LIN {X 0,Y 425.396,Z 103.811,A -85,B 0,C 180,E1 -9909.51,E2 -9909.51} C_VEL
LIN {X 0,Y 425.389,Z 103.807,A -85,B 0,C 180,E1 -9912.904,E2 -9912.904} C_VEL
LIN {X 0,Y 425.357,Z 103.809,A -85,B 0,C 180,E1 -9916.605,E2 -9916.605} C_VEL
LIN {X 0,Y 425.324,Z 103.816,A -85,B 0,C 180,E1 -9919.636,E2 -9919.636} C_VEL
LIN {X 0,Y 425.303,Z 103.821,A -85,B 0,C 180,E1 -9923.365,E2 -9923.365} C_VEL
LIN {X 0,Y 425.343,Z 103.814,A -85,B 0,C 180,E1 -9926.844,E2 -9926.844} C_VEL
LIN {X 0,Y 425.287,Z 103.819,A -85,B 0,C 180,E1 -9929.72,E2 -9929.72} C_VEL
LIN {X 0,Y 425.278,Z 103.826,A -85,B 0,C 180,E1 -9933.048,E2 -9933.048} C_VEL
LIN {X 0,Y 425.281,Z 103.818,A -85,B 0,C 180,E1 -9935.93,E2 -9935.93} C_VEL
LIN {X 0,Y 425.297,Z 103.823,A -85,B 0,C 180,E1 -9939.044,E2 -9939.044} C_VEL
LIN {X 0,Y 425.275,Z 103.824,A -85,B 0,C 180,E1 -9942.653,E2 -9942.653} C_VEL
LIN {X 0,Y 425.265,Z 103.821,A -85,B 0,C 180,E1 -9946.046,E2 -9946.046} C_VEL
LIN {X 0,Y 425.301,Z 103.821,A -85,B 0,C 180,E1 -9948.626,E2 -9948.626} C_VEL
LIN {X 0,Y 425.313,Z 103.818,A -85,B 0,C 180,E1 -9951.104,E2 -9951.104} C_VEL
LIN {X 0,Y 425.296,Z 103.824,A -85,B 0,C 180,E1 -9954.665,E2 -9954.665} C_VEL
LIN {X 0,Y 425.263,Z 103.822,A -85,B 0,C 180,E1 -9958.074,E2 -9958.074} C_VEL
LIN {X 0,Y 425.329,Z 103.813,A -85,B 0,C 180,E1 -9961.369,E2 -9961.369} C_VEL
LIN {X 0,Y 425.295,Z 103.824,A -85,B 0,C 180,E1 -9964.555,E2 -9964.555} C_VEL
LIN {X 0,Y 425.286,Z 103.818,A -85,B 0,C 180,E1 -9967.662,E2 -9967.662} C_VEL
LIN {X 0,Y 425.364,Z 103.812,A -85,B 0,C 180,E1 -9970.705,E2 -9970.705} C_VEL
LIN {X 0,Y 425.388,Z 103.806,A -85,B 0,C 180,E1 -9973.689,E2 -9973.689} C_VEL
LIN {X 0,Y 425.412,Z 103.803,A -85,B 0,C 180,E1 -9977.599,E2 -9977.599} C_VEL
LIN {X 0,Y 425.443,Z 103.799,A -85,B 0,C 180,E1 -9981.451,E2 -9981.451} C_VEL
LIN {X 0,Y 425.554,Z 103.79,A -85,B 0,C 180,E1 -9984.314,E2 -9984.314} C_VEL
LIN {X 0,Y 425.574,Z 103.79,A -85,B 0,C 180,E1 -9988.108,E2 -9988.108} C_VEL
LIN {X 0,Y 425.702,Z 103.773,A -85,B 0,C 180,E1 -9990.001,E2 -9990.001} C_VEL
LIN {X 0,Y 425.546,Z 103.786,A -85,B 0,C 180,E1 -9992.841,E2 -9992.841} C_VEL
LIN {X 0,Y 425.532,Z 103.788,A -85,B 0,C 180,E1 -9996.639,E2 -9996.639} C_VEL
LIN {X 0,Y 425.404,Z 103.804,A -85,B 0,C 180,E1 -9999.153,E2 -9999.153} C_VEL
LIN {X 0,Y 424.732,Z 103.894,A -85,B 0,C 180,E1 -9999.943,E2 -9999.943} C_VEL
LIN {X 0,Y 421.884,Z 104.243,A -85,B 0,C 180,E1 -10001.226,E2 -10001.226} C_VEL
LIN {X 0,Y 419.468,Z 104.545,A -85,B 0,C 180,E1 -10002.262,E2 -10002.262} C_VEL
LIN {X 0,Y 418.417,Z 104.674,A -85,B 0,C 180,E1 -10003.063,E2 -10003.063} C_VEL
LIN {X 0,Y 418.324,Z 104.687,A -85,B 0,C 180,E1 -10003.334,E2 -10003.334} C_VEL
LIN {X 0,Y 418.315,Z 104.686,A -85,B 0,C 180,E1 -10006.736,E2 -10006.736} C_VEL
LIN {X 0,Y 418.273,Z 104.698,A -85,B 0,C 180,E1 -10009.791,E2 -10009.791} C_VEL
LIN {X 0,Y 418.24,Z 104.696,A -85,B 0,C 180,E1 -10012.737,E2 -10012.737} C_VEL
LIN {X 0,Y 418.271,Z 104.695,A -85,B 0,C 180,E1 -10015.905,E2 -10015.905} C_VEL
LIN {X 0,Y 418.267,Z 104.695,A -85,B 0,C 180,E1 -10019.162,E2 -10019.162} C_VEL
LIN {X 0,Y 418.26,Z 104.694,A -85,B 0,C 180,E1 -10022.844,E2 -10022.844} C_VEL
LIN {X 0,Y 418.247,Z 104.695,A -85,B 0,C 180,E1 -10026.238,E2 -10026.238} C_VEL
LIN {X 0,Y 418.254,Z 104.697,A -85,B 0,C 180,E1 -10029.682,E2 -10029.682} C_VEL
LIN {X 0,Y 418.234,Z 104.696,A -85,B 0,C 180,E1 -10032.322,E2 -10032.322} C_VEL
LIN {X 0,Y 418.241,Z 104.701,A -85,B 0,C 180,E1 -10035.109,E2 -10035.109} C_VEL
LIN {X 0,Y 418.243,Z 104.697,A -85,B 0,C 180,E1 -10037.767,E2 -10037.767} C_VEL
LIN {X 0,Y 418.252,Z 104.696,A -85,B 0,C 180,E1 -10040.62,E2 -10040.62} C_VEL
LIN {X 0,Y 418.247,Z 104.699,A -85,B 0,C 180,E1 -10043.976,E2 -10043.976} C_VEL
LIN {X 0,Y 418.261,Z 104.698,A -85,B 0,C 180,E1 -10047.156,E2 -10047.156} C_VEL
LIN {X 0,Y 418.256,Z 104.744,A -85,B 0,C 180,E1 -10047.691,E2 -10047.691} C_VEL
LIN {X 0,Y 419.311,Z 107.662,A -85,B 0,C 180,E1 -10047.841,E2 -10047.841} C_VEL
LIN {X 0,Y 434.601,Z 137.945,A -85,B 0,C 180,E1 -10049.622,E2 -10049.622} C_VEL
LIN {X 0,Y 430.278,Z 282.426,A -85,B 0,C 180,E1 -10052.554,E2 -10052.554} C_VEL
LIN {X 0,Y 429.662,Z 301.528,A -85,B 0,C 180,E1 -10053.005,E2 -10053.005} C_VEL
LIN {X 0,Y 428.924,Z 318.826,A -85,B 0,C 180,E1 -10053.612,E2 -10053.612} C_VEL
LIN {X 0,Y 427.987,Z 335.334,A -85,B 0,C 180,E1 -10054.386,E2 -10054.386} C_VEL
LIN {X 0,Y 427.104,Z 349.564,A -85,B 0,C 180,E1 -10055.22,E2 -10055.22} C_VEL
LIN {X 0,Y 425.867,Z 364.452,A -85,B 0,C 180,E1 -10056.281,E2 -10056.281} C_VEL
LIN {X 0,Y 424.626,Z 378.646,A -85,B 0,C 180,E1 -10057.496,E2 -10057.496} C_VEL
LIN {X 0,Y 423.459,Z 391.882,A -85,B 0,C 180,E1 -10058.84,E2 -10058.84} C_VEL
LIN {X 0,Y 422.25,Z 404.22,A -85,B 0,C 180,E1 -10060.303,E2 -10060.303} C_VEL
LIN {X 0,Y 421.134,Z 416.557,A -85,B 0,C 180,E1 -10062.034,E2 -10062.034} C_VEL
LIN {X 0,Y 420.175,Z 426.779,A -85,B 0,C 180,E1 -10063.73,E2 -10063.73} C_VEL
LIN {X 0,Y 419.373,Z 435.593,A -85,B 0,C 180,E1 -10065.441,E2 -10065.441} C_VEL
LIN {X 0,Y 418.682,Z 444.113,A -85,B 0,C 180,E1 -10067.396,E2 -10067.396} C_VEL
LIN {X 0,Y 418.129,Z 451.181,A -85,B 0,C 180,E1 -10069.345,E2 -10069.345} C_VEL
LIN {X 0,Y 417.81,Z 456.853,A -85,B 0,C 180,E1 -10071.292,E2 -10071.292} C_VEL
LIN {X 0,Y 417.603,Z 461.379,A -85,B 0,C 180,E1 -10073.234,E2 -10073.234} C_VEL
LIN {X 0,Y 417.363,Z 464.808,A -85,B 0,C 180,E1 -10075.17,E2 -10075.17} C_VEL
LIN {X 0,Y 417.372,Z 467.119,A -85,B 0,C 180,E1 -10077.104,E2 -10077.104} C_VEL
LIN {X 0,Y 417.219,Z 468.502,A -85,B 0,C 180,E1 -10079.035,E2 -10079.035} C_VEL
LIN {X 0,Y 417.221,Z 468.775,A -85,B 0,C 180,E1 -10080.965,E2 -10080.965} C_VEL
LIN {X 0,Y 417.491,Z 468.097,A -85,B 0,C 180,E1 -10082.895,E2 -10082.895} C_VEL
LIN {X 0,Y 417.563,Z 466.374,A -85,B 0,C 180,E1 -10084.827,E2 -10084.827} C_VEL
LIN {X 0,Y 417.796,Z 463.165,A -85,B 0,C 180,E1 -10087.03,E2 -10087.03} C_VEL
LIN {X 0,Y 418.18,Z 458.676,A -85,B 0,C 180,E1 -10089.187,E2 -10089.187} C_VEL
LIN {X 0,Y 418.736,Z 453.445,A -85,B 0,C 180,E1 -10091.129,E2 -10091.129} C_VEL
LIN {X 0,Y 419.34,Z 446.871,A -85,B 0,C 180,E1 -10093.077,E2 -10093.077} C_VEL
LIN {X 0,Y 420.259,Z 438.912,A -85,B 0,C 180,E1 -10095.023,E2 -10095.023} C_VEL
LIN {X 0,Y 421.348,Z 429.335,A -85,B 0,C 180,E1 -10096.971,E2 -10096.971} C_VEL
LIN {X 0,Y 422.531,Z 419.574,A -85,B 0,C 180,E1 -10098.649,E2 -10098.649} C_VEL
LIN {X 0,Y 423.927,Z 407.703,A -85,B 0,C 180,E1 -10100.374,E2 -10100.374} C_VEL
LIN {X 0,Y 425.482,Z 393.99,A -85,B 0,C 180,E1 -10102.044,E2 -10102.044} C_VEL
LIN {X 0,Y 427.128,Z 379.392,A -85,B 0,C 180,E1 -10103.516,E2 -10103.516} C_VEL
LIN {X 0,Y 428.551,Z 365.071,A -85,B 0,C 180,E1 -10104.72,E2 -10104.72} C_VEL
LIN {X 0,Y 429.738,Z 351.619,A -85,B 0,C 180,E1 -10105.671,E2 -10105.671} C_VEL
LIN {X 0,Y 431.066,Z 334.858,A -85,B 0,C 180,E1 -10106.638,E2 -10106.638} C_VEL
LIN {X 0,Y 432.092,Z 318.332,A -85,B 0,C 180,E1 -10107.387,E2 -10107.387} C_VEL
LIN {X 0,Y 432.944,Z 301.612,A -85,B 0,C 180,E1 -10107.952,E2 -10107.952} C_VEL
LIN {X 0,Y 437.02,Z 225.54,A -85,B 0,C 180,E1 -10109.847,E2 -10109.847} C_VEL
LIN {X 0,Y 442.861,Z 147.406,A -85,B 0,C 180,E1 -10111.912,E2 -10111.912} C_VEL
LIN {X 0,Y 443.142,Z 143.294,A -85,B 0,C 180,E1 -10112.033,E2 -10112.033} C_VEL
LIN {X 0,Y 438.622,Z 134.82,A -85,B 0,C 180,E1 -10113.056,E2 -10113.056} C_VEL
LIN {X 0,Y 434.512,Z 127.988,A -85,B 0,C 180,E1 -10114.077,E2 -10114.077} C_VEL
LIN {X 0,Y 431.135,Z 123.216,A -85,B 0,C 180,E1 -10114.973,E2 -10114.973} C_VEL
LIN {X 0,Y 427.821,Z 118.988,A -85,B 0,C 180,E1 -10115.948,E2 -10115.948} C_VEL
LIN {X 0,Y 422.509,Z 113.054,A -85,B 0,C 180,E1 -10117.822,E2 -10117.822} C_VEL
LIN {X 0,Y 421.55,Z 111.994,A -85,B 0,C 180,E1 -10118.3,E2 -10118.3} C_VEL
LIN {X 0,Y 420.598,Z 109.865,A -85,B 0,C 180,E1 -10120.668,E2 -10120.668} C_VEL
LIN {X 0,Y 420.52,Z 109.347,A -85,B 0,C 180,E1 -10121.952,E2 -10121.952} C_VEL
LIN {X 0,Y 420.653,Z 110.069,A -85,B 0,C 180,E1 -10124.075,E2 -10124.075} C_VEL
LIN {X 0,Y 421.369,Z 111.749,A -85,B 0,C 180,E1 -10125.823,E2 -10125.823} C_VEL
LIN {X 0,Y 422.878,Z 114.606,A -85,B 0,C 180,E1 -10127.738,E2 -10127.738} C_VEL
LIN {X 0,Y 424.752,Z 118.675,A -85,B 0,C 180,E1 -10129.563,E2 -10129.563} C_VEL
LIN {X 0,Y 426.873,Z 123.698,A -85,B 0,C 180,E1 -10131.271,E2 -10131.271} C_VEL
LIN {X 0,Y 429.708,Z 131.075,A -85,B 0,C 180,E1 -10133.264,E2 -10133.264} C_VEL
LIN {X 0,Y 431.088,Z 134.99,A -85,B 0,C 180,E1 -10134.126,E2 -10134.126} C_VEL
LIN {X 0,Y 435.256,Z 143.345,A -85,B 0,C 180,E1 -10135.282,E2 -10135.282} C_VEL
LIN {X 0,Y 437.837,Z 149.267,A -85,B 0,C 180,E1 -10135.963,E2 -10135.963} C_VEL
LIN {X 0,Y 439.521,Z 164.422,A -85,B 0,C 180,E1 -10136.829,E2 -10136.829} C_VEL
LIN {X 0,Y 440.924,Z 183.827,A -85,B 0,C 180,E1 -10137.748,E2 -10137.748} C_VEL
LIN {X 0,Y 441.044,Z 188.8,A -85,B 0,C 180,E1 -10137.944,E2 -10137.944} C_VEL
LIN {X 0,Y 436.113,Z 262.024,A -85,B 0,C 180,E1 -10139.828,E2 -10139.828} C_VEL
LIN {X 0,Y 432.849,Z 326.235,A -85,B 0,C 180,E1 -10141.39,E2 -10141.39} C_VEL
LIN {X 0,Y 431.402,Z 356.177,A -85,B 0,C 180,E1 -10142.137,E2 -10142.137} C_VEL
LIN {X 0,Y 429.892,Z 374.913,A -85,B 0,C 180,E1 -10142.79,E2 -10142.79} C_VEL
LIN {X 0,Y 428.455,Z 391.774,A -85,B 0,C 180,E1 -10143.58,E2 -10143.58} C_VEL
LIN {X 0,Y 426.854,Z 407.978,A -85,B 0,C 180,E1 -10144.523,E2 -10144.523} C_VEL
LIN {X 0,Y 425.144,Z 424.654,A -85,B 0,C 180,E1 -10145.719,E2 -10145.719} C_VEL
LIN {X 0,Y 423.574,Z 440.021,A -85,B 0,C 180,E1 -10147.05,E2 -10147.05} C_VEL
LIN {X 0,Y 422.113,Z 454.241,A -85,B 0,C 180,E1 -10148.512,E2 -10148.512} C_VEL
LIN {X 0,Y 420.719,Z 468.305,A -85,B 0,C 180,E1 -10150.228,E2 -10150.228} C_VEL
LIN {X 0,Y 419.628,Z 480.238,A -85,B 0,C 180,E1 -10151.95,E2 -10151.95} C_VEL
LIN {X 0,Y 418.772,Z 490.482,A -85,B 0,C 180,E1 -10153.673,E2 -10153.673} C_VEL
LIN {X 0,Y 418.162,Z 499.345,A -85,B 0,C 180,E1 -10155.397,E2 -10155.397} C_VEL
LIN {X 0,Y 417.694,Z 507.935,A -85,B 0,C 180,E1 -10157.392,E2 -10157.392} C_VEL
LIN {X 0,Y 417.361,Z 514.845,A -85,B 0,C 180,E1 -10159.325,E2 -10159.325} C_VEL
LIN {X 0,Y 417.231,Z 520.598,A -85,B 0,C 180,E1 -10161.28,E2 -10161.28} C_VEL
LIN {X 0,Y 417.307,Z 525.707,A -85,B 0,C 180,E1 -10163.531,E2 -10163.531} C_VEL
LIN {X 0,Y 417.187,Z 529.663,A -85,B 0,C 180,E1 -10166.136,E2 -10166.136} C_VEL
LIN {X 0,Y 417.281,Z 531.295,A -85,B 0,C 180,E1 -10168.069,E2 -10168.069} C_VEL
LIN {X 0,Y 417.174,Z 531.882,A -85,B 0,C 180,E1 -10169.999,E2 -10169.999} C_VEL
LIN {X 0,Y 417.294,Z 531.377,A -85,B 0,C 180,E1 -10171.93,E2 -10171.93} C_VEL
LIN {X 0,Y 417.191,Z 529.776,A -85,B 0,C 180,E1 -10173.863,E2 -10173.863} C_VEL
LIN {X 0,Y 417.217,Z 527.105,A -85,B 0,C 180,E1 -10175.8,E2 -10175.8} C_VEL
LIN {X 0,Y 417.222,Z 523.234,A -85,B 0,C 180,E1 -10177.744,E2 -10177.744} C_VEL
LIN {X 0,Y 417.231,Z 518.213,A -85,B 0,C 180,E1 -10179.697,E2 -10179.697} C_VEL
LIN {X 0,Y 417.51,Z 511.87,A -85,B 0,C 180,E1 -10181.653,E2 -10181.653} C_VEL
LIN {X 0,Y 417.894,Z 504.094,A -85,B 0,C 180,E1 -10183.617,E2 -10183.617} C_VEL
LIN {X 0,Y 418.57,Z 494.75,A -85,B 0,C 180,E1 -10185.583,E2 -10185.583} C_VEL
LIN {X 0,Y 419.329,Z 484.83,A -85,B 0,C 180,E1 -10187.349,E2 -10187.349} C_VEL
LIN {X 0,Y 420.25,Z 473.712,A -85,B 0,C 180,E1 -10189.032,E2 -10189.032} C_VEL
LIN {X 0,Y 421.454,Z 461.108,A -85,B 0,C 180,E1 -10190.648,E2 -10190.648} C_VEL
LIN {X 0,Y 422.725,Z 447.832,A -85,B 0,C 180,E1 -10192.095,E2 -10192.095} C_VEL
LIN {X 0,Y 424.021,Z 433.225,A -85,B 0,C 180,E1 -10193.439,E2 -10193.439} C_VEL
LIN {X 0,Y 425.488,Z 417.781,A -85,B 0,C 180,E1 -10194.615,E2 -10194.615} C_VEL
LIN {X 0,Y 426.713,Z 402.934,A -85,B 0,C 180,E1 -10195.55,E2 -10195.55} C_VEL
LIN {X 0,Y 427.953,Z 386.241,A -85,B 0,C 180,E1 -10196.386,E2 -10196.386} C_VEL
LIN {X 0,Y 429.007,Z 368.899,A -85,B 0,C 180,E1 -10197.038,E2 -10197.038} C_VEL
LIN {X 0,Y 429.847,Z 351.558,A -85,B 0,C 180,E1 -10197.487,E2 -10197.487} C_VEL
LIN {X 0,Y 434.839,Z 186.692,A -85,B 0,C 180,E1 -10200.839,E2 -10200.839} C_VEL
LIN {X 0,Y 429.925,Z 149.859,A -85,B 0,C 180,E1 -10202.053,E2 -10202.053} C_VEL
LIN {X 0,Y 430.466,Z 143.061,A -85,B 0,C 180,E1 -10202.756,E2 -10202.756} C_VEL
LIN {X 0,Y 426.121,Z 128.649,A -85,B 0,C 180,E1 -10204.656,E2 -10204.656} C_VEL
LIN {X 0,Y 419.021,Z 107.167,A -85,B 0,C 180,E1 -10207.659,E2 -10207.659} C_VEL
LIN {X 0,Y 418.224,Z 104.704,A -85,B 0,C 180,E1 -10208.033,E2 -10208.033} C_VEL
LIN {X 0,Y 418.257,Z 104.699,A -85,B 0,C 180,E1 -10210.943,E2 -10210.943} C_VEL
LIN {X 0,Y 418.264,Z 104.696,A -85,B 0,C 180,E1 -10213.737,E2 -10213.737} C_VEL
LIN {X 0,Y 418.207,Z 104.706,A -85,B 0,C 180,E1 -10216.449,E2 -10216.449} C_VEL
LIN {X 0,Y 418.22,Z 104.698,A -85,B 0,C 180,E1 -10219.13,E2 -10219.13} C_VEL
LIN {X 0,Y 418.23,Z 104.703,A -85,B 0,C 180,E1 -10222.165,E2 -10222.165} C_VEL
LIN {X 0,Y 418.261,Z 104.693,A -85,B 0,C 180,E1 -10225.419,E2 -10225.419} C_VEL
LIN {X 0,Y 418.215,Z 104.701,A -85,B 0,C 180,E1 -10228.604,E2 -10228.604} C_VEL
LIN {X 0,Y 418.29,Z 104.694,A -85,B 0,C 180,E1 -10231.937,E2 -10231.937} C_VEL
LIN {X 0,Y 418.285,Z 104.69,A -85,B 0,C 180,E1 -10235.163,E2 -10235.163} C_VEL
LIN {X 0,Y 418.23,Z 104.701,A -85,B 0,C 180,E1 -10238.304,E2 -10238.304} C_VEL
LIN {X 0,Y 418.279,Z 104.692,A -85,B 0,C 180,E1 -10241.383,E2 -10241.383} C_VEL
LIN {X 0,Y 418.306,Z 104.689,A -85,B 0,C 180,E1 -10244.406,E2 -10244.406} C_VEL
LIN {X 0,Y 418.365,Z 104.682,A -85,B 0,C 180,E1 -10247.386,E2 -10247.386} C_VEL
LIN {X 0,Y 418.355,Z 104.683,A -85,B 0,C 180,E1 -10250.329,E2 -10250.329} C_VEL
LIN {X 0,Y 418.489,Z 104.666,A -85,B 0,C 180,E1 -10253.249,E2 -10253.249} C_VEL
LIN {X 0,Y 418.336,Z 104.685,A -85,B 0,C 180,E1 -10255.182,E2 -10255.182} C_VEL
LIN {X 0,Y 418.54,Z 104.661,A -85,B 0,C 180,E1 -10258.076,E2 -10258.076} C_VEL
LIN {X 0,Y 418.668,Z 104.645,A -85,B 0,C 180,E1 -10260,E2 -10260} C_VEL
LIN {X 0,Y 418.506,Z 104.663,A -85,B 0,C 180,E1 -10262.888,E2 -10262.888} C_VEL
LIN {X 0,Y 418.489,Z 104.665,A -85,B 0,C 180,E1 -10266.751,E2 -10266.751} C_VEL
LIN {X 0,Y 418.396,Z 104.677,A -85,B 0,C 180,E1 -10268.695,E2 -10268.695} C_VEL
LIN {X 0,Y 418.312,Z 104.691,A -85,B 0,C 180,E1 -10271.631,E2 -10271.631} C_VEL
LIN {X 0,Y 418.299,Z 104.689,A -85,B 0,C 180,E1 -10274.597,E2 -10274.597} C_VEL
LIN {X 0,Y 418.284,Z 104.694,A -85,B 0,C 180,E1 -10277.604,E2 -10277.604} C_VEL
LIN {X 0,Y 418.246,Z 104.696,A -85,B 0,C 180,E1 -10280.663,E2 -10280.663} C_VEL
LIN {X 0,Y 418.284,Z 104.692,A -85,B 0,C 180,E1 -10283.781,E2 -10283.781} C_VEL
LIN {X 0,Y 418.306,Z 104.694,A -85,B 0,C 180,E1 -10287.071,E2 -10287.071} C_VEL
LIN {X 0,Y 418.24,Z 104.696,A -85,B 0,C 180,E1 -10290.272,E2 -10290.272} C_VEL
LIN {X 0,Y 418.245,Z 104.696,A -85,B 0,C 180,E1 -10293.677,E2 -10293.677} C_VEL
LIN {X 0,Y 418.242,Z 104.7,A -85,B 0,C 180,E1 -10297.224,E2 -10297.224} C_VEL
LIN {X 0,Y 418.249,Z 104.695,A -85,B 0,C 180,E1 -10299.682,E2 -10299.682} C_VEL
LIN {X 0,Y 418.229,Z 104.698,A -85,B 0,C 180,E1 -10302.322,E2 -10302.322} C_VEL
LIN {X 0,Y 418.239,Z 104.7,A -85,B 0,C 180,E1 -10305.11,E2 -10305.11} C_VEL
LIN {X 0,Y 418.255,Z 104.694,A -85,B 0,C 180,E1 -10307.77,E2 -10307.77} C_VEL
LIN {X 0,Y 418.26,Z 104.699,A -85,B 0,C 180,E1 -10310.618,E2 -10310.618} C_VEL
LIN {X 0,Y 418.24,Z 104.696,A -85,B 0,C 180,E1 -10313.976,E2 -10313.976} C_VEL
LIN {X 0,Y 418.255,Z 104.695,A -85,B 0,C 180,E1 -10317.157,E2 -10317.157} C_VEL
LIN {X 0,Y 418.266,Z 104.696,A -85,B 0,C 180,E1 -10320.896,E2 -10320.896} C_VEL
LIN {X 0,Y 418.27,Z 104.694,A -85,B 0,C 180,E1 -10324.097,E2 -10324.097} C_VEL
LIN {X 0,Y 418.237,Z 104.696,A -85,B 0,C 180,E1 -10327.265,E2 -10327.265} C_VEL
LIN {X 0,Y 418.315,Z 104.693,A -85,B 0,C 180,E1 -10330.366,E2 -10330.366} C_VEL
LIN {X 0,Y 418.316,Z 104.686,A -85,B 0,C 180,E1 -10333.405,E2 -10333.405} C_VEL
LIN {X 0,Y 418.346,Z 104.683,A -85,B 0,C 180,E1 -10337,E2 -10337} C_VEL
LIN {X 0,Y 418.357,Z 104.687,A -85,B 0,C 180,E1 -10340.33,E2 -10340.33} C_VEL
LIN {X 0,Y 418.494,Z 104.664,A -85,B 0,C 180,E1 -10343.25,E2 -10343.25} C_VEL
LIN {X 0,Y 418.339,Z 104.683,A -85,B 0,C 180,E1 -10345.182,E2 -10345.182} C_VEL
LIN {X 0,Y 418.543,Z 104.665,A -85,B 0,C 180,E1 -10348.076,E2 -10348.076} C_VEL
LIN {X 0,Y 418.671,Z 104.649,A -85,B 0,C 180,E1 -10350.001,E2 -10350.001} C_VEL
LIN {X 0,Y 418.502,Z 104.663,A -85,B 0,C 180,E1 -10352.888,E2 -10352.888} C_VEL
LIN {X 0,Y 418.495,Z 104.664,A -85,B 0,C 180,E1 -10356.752,E2 -10356.752} C_VEL
LIN {X 0,Y 418.359,Z 104.681,A -85,B 0,C 180,E1 -10359.144,E2 -10359.144} C_VEL
LIN {X 0,Y 418.357,Z 104.681,A -85,B 0,C 180,E1 -10362.615,E2 -10362.615} C_VEL
LIN {X 0,Y 418.324,Z 104.687,A -85,B 0,C 180,E1 -10363.334,E2 -10363.334} C_VEL
LIN {X 0,Y 417.63,Z 104.778,A -85,B 0,C 180,E1 -10364.138,E2 -10364.138} C_VEL
LIN {X 0,Y 414.752,Z 105.133,A -85,B 0,C 180,E1 -10365.443,E2 -10365.443} C_VEL
LIN {X 0,Y 412.34,Z 105.431,A -85,B 0,C 180,E1 -10366.497,E2 -10366.497} C_VEL
LIN {X 0,Y 411.318,Z 105.56,A -85,B 0,C 180,E1 -10367.312,E2 -10367.312} C_VEL
LIN {X 0,Y 411.242,Z 105.569,A -85,B 0,C 180,E1 -10367.588,E2 -10367.588} C_VEL
LIN {X 0,Y 411.199,Z 105.574,A -85,B 0,C 180,E1 -10371.035,E2 -10371.035} C_VEL
LIN {X 0,Y 411.227,Z 105.57,A -85,B 0,C 180,E1 -10374.216,E2 -10374.216} C_VEL
LIN {X 0,Y 411.261,Z 105.571,A -85,B 0,C 180,E1 -10377.478,E2 -10377.478} C_VEL
LIN {X 0,Y 411.192,Z 105.574,A -85,B 0,C 180,E1 -10380.848,E2 -10380.848} C_VEL
LIN {X 0,Y 411.208,Z 105.572,A -85,B 0,C 180,E1 -10384.334,E2 -10384.334} C_VEL
LIN {X 0,Y 411.198,Z 105.574,A -85,B 0,C 180,E1 -10387.974,E2 -10387.974} C_VEL
LIN {X 0,Y 411.184,Z 105.575,A -85,B 0,C 180,E1 -10390.505,E2 -10390.505} C_VEL
LIN {X 0,Y 411.18,Z 105.58,A -85,B 0,C 180,E1 -10393.133,E2 -10393.133} C_VEL
LIN {X 0,Y 411.171,Z 105.577,A -85,B 0,C 180,E1 -10395.881,E2 -10395.881} C_VEL
LIN {X 0,Y 411.166,Z 105.579,A -85,B 0,C 180,E1 -10398.772,E2 -10398.772} C_VEL
LIN {X 0,Y 411.196,Z 105.573,A -85,B 0,C 180,E1 -10402.026,E2 -10402.026} C_VEL
LIN {X 0,Y 411.209,Z 105.575,A -85,B 0,C 180,E1 -10405.667,E2 -10405.667} C_VEL
LIN {X 0,Y 411.236,Z 105.733,A -85,B 0,C 180,E1 -10407.193,E2 -10407.193} C_VEL
LIN {X 0,Y 412.352,Z 108.62,A -85,B 0,C 180,E1 -10407.349,E2 -10407.349} C_VEL
LIN {X 0,Y 428.152,Z 140.061,A -85,B 0,C 180,E1 -10409.238,E2 -10409.238} C_VEL
LIN {X 0,Y 424.246,Z 262.856,A -85,B 0,C 180,E1 -10411.794,E2 -10411.794} C_VEL
LIN {X 0,Y 423.261,Z 297.329,A -85,B 0,C 180,E1 -10412.529,E2 -10412.529} C_VEL
LIN {X 0,Y 422.59,Z 314.428,A -85,B 0,C 180,E1 -10413.085,E2 -10413.085} C_VEL
LIN {X 0,Y 421.688,Z 330.419,A -85,B 0,C 180,E1 -10413.79,E2 -10413.79} C_VEL
LIN {X 0,Y 420.668,Z 345.765,A -85,B 0,C 180,E1 -10414.648,E2 -10414.648} C_VEL
LIN {X 0,Y 419.391,Z 361.884,A -85,B 0,C 180,E1 -10415.76,E2 -10415.76} C_VEL
LIN {X 0,Y 418.054,Z 376.619,A -85,B 0,C 180,E1 -10416.992,E2 -10416.992} C_VEL
LIN {X 0,Y 416.799,Z 390.284,A -85,B 0,C 180,E1 -10418.355,E2 -10418.355} C_VEL
LIN {X 0,Y 415.692,Z 401.907,A -85,B 0,C 180,E1 -10419.721,E2 -10419.721} C_VEL
LIN {X 0,Y 414.565,Z 412.871,A -85,B 0,C 180,E1 -10421.21,E2 -10421.21} C_VEL
LIN {X 0,Y 413.569,Z 423.875,A -85,B 0,C 180,E1 -10422.954,E2 -10422.954} C_VEL
LIN {X 0,Y 412.52,Z 434.461,A -85,B 0,C 180,E1 -10424.941,E2 -10424.941} C_VEL
LIN {X 0,Y 411.855,Z 442.507,A -85,B 0,C 180,E1 -10426.746,E2 -10426.746} C_VEL
LIN {X 0,Y 411.222,Z 449.701,A -85,B 0,C 180,E1 -10428.665,E2 -10428.665} C_VEL
LIN {X 0,Y 410.844,Z 455.842,A -85,B 0,C 180,E1 -10430.647,E2 -10430.647} C_VEL
LIN {X 0,Y 410.586,Z 460.722,A -85,B 0,C 180,E1 -10432.624,E2 -10432.624} C_VEL
LIN {X 0,Y 410.403,Z 463.66,A -85,B 0,C 180,E1 -10434.102,E2 -10434.102} C_VEL
LIN {X 0,Y 410.366,Z 466.536,A -85,B 0,C 180,E1 -10436.072,E2 -10436.072} C_VEL
LIN {X 0,Y 410.267,Z 468.445,A -85,B 0,C 180,E1 -10438.037,E2 -10438.037} C_VEL
LIN {X 0,Y 410.134,Z 469.315,A -85,B 0,C 180,E1 -10440,E2 -10440} C_VEL
LIN {X 0,Y 410.275,Z 469.161,A -85,B 0,C 180,E1 -10441.963,E2 -10441.963} C_VEL
LIN {X 0,Y 410.45,Z 468.021,A -85,B 0,C 180,E1 -10443.927,E2 -10443.927} C_VEL
LIN {X 0,Y 410.467,Z 465.825,A -85,B 0,C 180,E1 -10445.896,E2 -10445.896} C_VEL
LIN {X 0,Y 410.92,Z 462.616,A -85,B 0,C 180,E1 -10447.864,E2 -10447.864} C_VEL
LIN {X 0,Y 411.473,Z 456.988,A -85,B 0,C 180,E1 -10450.331,E2 -10450.331} C_VEL
LIN {X 0,Y 412.09,Z 451.128,A -85,B 0,C 180,E1 -10452.309,E2 -10452.309} C_VEL
LIN {X 0,Y 413.023,Z 443.048,A -85,B 0,C 180,E1 -10454.511,E2 -10454.511} C_VEL
LIN {X 0,Y 414.17,Z 434.037,A -85,B 0,C 180,E1 -10456.513,E2 -10456.513} C_VEL
LIN {X 0,Y 415.363,Z 424.388,A -85,B 0,C 180,E1 -10458.319,E2 -10458.319} C_VEL
LIN {X 0,Y 416.748,Z 414.01,A -85,B 0,C 180,E1 -10459.968,E2 -10459.968} C_VEL
LIN {X 0,Y 418.263,Z 401.201,A -85,B 0,C 180,E1 -10461.695,E2 -10461.695} C_VEL
LIN {X 0,Y 420.042,Z 387.332,A -85,B 0,C 180,E1 -10463.244,E2 -10463.244} C_VEL
LIN {X 0,Y 421.632,Z 372.637,A -85,B 0,C 180,E1 -10464.627,E2 -10464.627} C_VEL
LIN {X 0,Y 423.225,Z 356.758,A -85,B 0,C 180,E1 -10465.857,E2 -10465.857} C_VEL
LIN {X 0,Y 424.724,Z 340.541,A -85,B 0,C 180,E1 -10466.868,E2 -10466.868} C_VEL
LIN {X 0,Y 425.894,Z 323.529,A -85,B 0,C 180,E1 -10467.719,E2 -10467.719} C_VEL
LIN {X 0,Y 426.961,Z 305.819,A -85,B 0,C 180,E1 -10468.379,E2 -10468.379} C_VEL
LIN {X 0,Y 428.53,Z 275.41,A -85,B 0,C 180,E1 -10469.169,E2 -10469.169} C_VEL
LIN {X 0,Y 432.99,Z 207.451,A -85,B 0,C 180,E1 -10470.952,E2 -10470.952} C_VEL
LIN {X 0,Y 438.134,Z 146.313,A -85,B 0,C 180,E1 -10472.644,E2 -10472.644} C_VEL
LIN {X 0,Y 433.199,Z 137.027,A -85,B 0,C 180,E1 -10473.876,E2 -10473.876} C_VEL
LIN {X 0,Y 429.427,Z 131.063,A -85,B 0,C 180,E1 -10474.897,E2 -10474.897} C_VEL
LIN {X 0,Y 425.187,Z 125.347,A -85,B 0,C 180,E1 -10476.185,E2 -10476.185} C_VEL
LIN {X 0,Y 420.318,Z 119.723,A -85,B 0,C 180,E1 -10477.975,E2 -10477.975} C_VEL
LIN {X 0,Y 416.442,Z 116.083,A -85,B 0,C 180,E1 -10479.888,E2 -10479.888} C_VEL
LIN {X 0,Y 415.786,Z 115.206,A -85,B 0,C 180,E1 -10480.479,E2 -10480.479} C_VEL
LIN {X 0,Y 415.735,Z 114.58,A -85,B 0,C 180,E1 -10481.941,E2 -10481.941} C_VEL
LIN {X 0,Y 415.821,Z 115.175,A -85,B 0,C 180,E1 -10483.865,E2 -10483.865} C_VEL
LIN {X 0,Y 416.838,Z 117.555,A -85,B 0,C 180,E1 -10486.269,E2 -10486.269} C_VEL
LIN {X 0,Y 418.047,Z 119.844,A -85,B 0,C 180,E1 -10487.742,E2 -10487.742} C_VEL
LIN {X 0,Y 419.89,Z 123.959,A -85,B 0,C 180,E1 -10489.601,E2 -10489.601} C_VEL
LIN {X 0,Y 422.142,Z 129.545,A -85,B 0,C 180,E1 -10491.487,E2 -10491.487} C_VEL
LIN {X 0,Y 423.279,Z 132.399,A -85,B 0,C 180,E1 -10492.247,E2 -10492.247} C_VEL
LIN {X 0,Y 428.06,Z 141.31,A -85,B 0,C 180,E1 -10493.855,E2 -10493.855} C_VEL
LIN {X 0,Y 431.394,Z 148.338,A -85,B 0,C 180,E1 -10494.852,E2 -10494.852} C_VEL
LIN {X 0,Y 433.409,Z 153.136,A -85,B 0,C 180,E1 -10495.42,E2 -10495.42} C_VEL
LIN {X 0,Y 434.932,Z 169.745,A -85,B 0,C 180,E1 -10496.381,E2 -10496.381} C_VEL
LIN {X 0,Y 435.968,Z 188.427,A -85,B 0,C 180,E1 -10497.27,E2 -10497.27} C_VEL
LIN {X 0,Y 430.755,Z 259.475,A -85,B 0,C 180,E1 -10499.175,E2 -10499.175} C_VEL
LIN {X 0,Y 426.985,Z 326.119,A -85,B 0,C 180,E1 -10500.854,E2 -10500.854} C_VEL
LIN {X 0,Y 425.423,Z 355.392,A -85,B 0,C 180,E1 -10501.61,E2 -10501.61} C_VEL
LIN {X 0,Y 423.842,Z 373.838,A -85,B 0,C 180,E1 -10502.268,E2 -10502.268} C_VEL
LIN {X 0,Y 422.464,Z 388.98,A -85,B 0,C 180,E1 -10502.975,E2 -10502.975} C_VEL
LIN {X 0,Y 420.646,Z 406.331,A -85,B 0,C 180,E1 -10503.986,E2 -10503.986} C_VEL
LIN {X 0,Y 418.794,Z 423.076,A -85,B 0,C 180,E1 -10505.194,E2 -10505.194} C_VEL
LIN {X 0,Y 417.124,Z 438.528,A -85,B 0,C 180,E1 -10506.543,E2 -10506.543} C_VEL
LIN {X 0,Y 415.533,Z 452.788,A -85,B 0,C 180,E1 -10508.024,E2 -10508.024} C_VEL
LIN {X 0,Y 414.103,Z 465.99,A -85,B 0,C 180,E1 -10509.639,E2 -10509.639} C_VEL
LIN {X 0,Y 412.879,Z 478.173,A -85,B 0,C 180,E1 -10511.387,E2 -10511.387} C_VEL
LIN {X 0,Y 411.931,Z 488.647,A -85,B 0,C 180,E1 -10513.139,E2 -10513.139} C_VEL
LIN {X 0,Y 411.163,Z 498.836,A -85,B 0,C 180,E1 -10515.143,E2 -10515.143} C_VEL
LIN {X 0,Y 410.638,Z 507.946,A -85,B 0,C 180,E1 -10517.301,E2 -10517.301} C_VEL
LIN {X 0,Y 410.218,Z 515.915,A -85,B 0,C 180,E1 -10519.636,E2 -10519.636} C_VEL
LIN {X 0,Y 410.142,Z 521.277,A -85,B 0,C 180,E1 -10521.624,E2 -10521.624} C_VEL
LIN {X 0,Y 410.218,Z 525.41,A -85,B 0,C 180,E1 -10523.551,E2 -10523.551} C_VEL
LIN {X 0,Y 410.095,Z 529.12,A -85,B 0,C 180,E1 -10526.069,E2 -10526.069} C_VEL
LIN {X 0,Y 410.198,Z 530.751,A -85,B 0,C 180,E1 -10528.036,E2 -10528.036} C_VEL
LIN {X 0,Y 410.118,Z 531.317,A -85,B 0,C 180,E1 -10529.999,E2 -10529.999} C_VEL
LIN {X 0,Y 410.223,Z 530.8,A -85,B 0,C 180,E1 -10531.963,E2 -10531.963} C_VEL
LIN {X 0,Y 410.103,Z 529.156,A -85,B 0,C 180,E1 -10533.93,E2 -10533.93} C_VEL
LIN {X 0,Y 410.152,Z 526.463,A -85,B 0,C 180,E1 -10535.9,E2 -10535.9} C_VEL
LIN {X 0,Y 410.14,Z 522.533,A -85,B 0,C 180,E1 -10537.879,E2 -10537.879} C_VEL
LIN {X 0,Y 410.162,Z 517.446,A -85,B 0,C 180,E1 -10539.865,E2 -10539.865} C_VEL
LIN {X 0,Y 410.471,Z 511.061,A -85,B 0,C 180,E1 -10541.856,E2 -10541.856} C_VEL
LIN {X 0,Y 410.883,Z 503.201,A -85,B 0,C 180,E1 -10543.854,E2 -10543.854} C_VEL
LIN {X 0,Y 411.552,Z 493.753,A -85,B 0,C 180,E1 -10545.856,E2 -10545.856} C_VEL
LIN {X 0,Y 412.348,Z 483.657,A -85,B 0,C 180,E1 -10547.661,E2 -10547.661} C_VEL
LIN {X 0,Y 413.357,Z 472.505,A -85,B 0,C 180,E1 -10549.362,E2 -10549.362} C_VEL
LIN {X 0,Y 414.633,Z 459.76,A -85,B 0,C 180,E1 -10551.004,E2 -10551.004} C_VEL
LIN {X 0,Y 415.952,Z 446.291,A -85,B 0,C 180,E1 -10552.474,E2 -10552.474} C_VEL
LIN {X 0,Y 417.201,Z 432.913,A -85,B 0,C 180,E1 -10553.714,E2 -10553.714} C_VEL
LIN {X 0,Y 418.68,Z 417.77,A -85,B 0,C 180,E1 -10554.889,E2 -10554.889} C_VEL
LIN {X 0,Y 419.99,Z 402.703,A -85,B 0,C 180,E1 -10555.856,E2 -10555.856} C_VEL
LIN {X 0,Y 421.258,Z 386.072,A -85,B 0,C 180,E1 -10556.705,E2 -10556.705} C_VEL
LIN {X 0,Y 422.354,Z 368.892,A -85,B 0,C 180,E1 -10557.366,E2 -10557.366} C_VEL
LIN {X 0,Y 423.198,Z 352.013,A -85,B 0,C 180,E1 -10557.819,E2 -10557.819} C_VEL
LIN {X 0,Y 428.426,Z 186.805,A -85,B 0,C 180,E1 -10561.262,E2 -10561.262} C_VEL
LIN {X 0,Y 423.48,Z 149.466,A -85,B 0,C 180,E1 -10562.524,E2 -10562.524} C_VEL
LIN {X 0,Y 423.754,Z 144.641,A -85,B 0,C 180,E1 -10563.04,E2 -10563.04} C_VEL
LIN {X 0,Y 418.264,Z 126.994,A -85,B 0,C 180,E1 -10565.42,E2 -10565.42} C_VEL
LIN {X 0,Y 411.226,Z 105.576,A -85,B 0,C 180,E1 -10568.51,E2 -10568.51} C_VEL
LIN {X 0,Y 411.214,Z 105.576,A -85,B 0,C 180,E1 -10571.8,E2 -10571.8} C_VEL
LIN {X 0,Y 411.219,Z 105.577,A -85,B 0,C 180,E1 -10574.483,E2 -10574.483} C_VEL
LIN {X 0,Y 411.173,Z 105.581,A -85,B 0,C 180,E1 -10578.194,E2 -10578.194} C_VEL
LIN {X 0,Y 411.219,Z 105.572,A -85,B 0,C 180,E1 -10580.776,E2 -10580.776} C_VEL
LIN {X 0,Y 411.195,Z 105.578,A -85,B 0,C 180,E1 -10584.471,E2 -10584.471} C_VEL
LIN {X 0,Y 411.166,Z 105.582,A -85,B 0,C 180,E1 -10588.003,E2 -10588.003} C_VEL
LIN {X 0,Y 411.218,Z 105.571,A -85,B 0,C 180,E1 -10591.41,E2 -10591.41} C_VEL
LIN {X 0,Y 411.232,Z 105.57,A -85,B 0,C 180,E1 -10594.707,E2 -10594.707} C_VEL
LIN {X 0,Y 411.201,Z 105.578,A -85,B 0,C 180,E1 -10597.913,E2 -10597.913} C_VEL
LIN {X 0,Y 411.22,Z 105.57,A -85,B 0,C 180,E1 -10601.051,E2 -10601.051} C_VEL
LIN {X 0,Y 411.258,Z 105.57,A -85,B 0,C 180,E1 -10604.132,E2 -10604.132} C_VEL
LIN {X 0,Y 411.31,Z 105.56,A -85,B 0,C 180,E1 -10607.166,E2 -10607.166} C_VEL
LIN {X 0,Y 411.303,Z 105.563,A -85,B 0,C 180,E1 -10610.162,E2 -10610.162} C_VEL
LIN {X 0,Y 411.456,Z 105.542,A -85,B 0,C 180,E1 -10613.133,E2 -10613.133} C_VEL
LIN {X 0,Y 411.307,Z 105.56,A -85,B 0,C 180,E1 -10615.099,E2 -10615.099} C_VEL
LIN {X 0,Y 411.509,Z 105.537,A -85,B 0,C 180,E1 -10618.043,E2 -10618.043} C_VEL
LIN {X 0,Y 411.638,Z 105.521,A -85,B 0,C 180,E1 -10620,E2 -10620} C_VEL
LIN {X 0,Y 411.462,Z 105.541,A -85,B 0,C 180,E1 -10622.937,E2 -10622.937} C_VEL
LIN {X 0,Y 411.456,Z 105.542,A -85,B 0,C 180,E1 -10626.867,E2 -10626.867} C_VEL
LIN {X 0,Y 411.288,Z 105.564,A -85,B 0,C 180,E1 -10629.839,E2 -10629.839} C_VEL
LIN {X 0,Y 411.301,Z 105.564,A -85,B 0,C 180,E1 -10633.104,E2 -10633.104} C_VEL
LIN {X 0,Y 411.258,Z 105.567,A -85,B 0,C 180,E1 -10636.869,E2 -10636.869} C_VEL
LIN {X 0,Y 411.226,Z 105.57,A -85,B 0,C 180,E1 -10639.987,E2 -10639.987} C_VEL
LIN {X 0,Y 411.199,Z 105.579,A -85,B 0,C 180,E1 -10643.148,E2 -10643.148} C_VEL
LIN {X 0,Y 411.234,Z 105.569,A -85,B 0,C 180,E1 -10646.381,E2 -10646.381} C_VEL
LIN {X 0,Y 411.196,Z 105.574,A -85,B 0,C 180,E1 -10649.713,E2 -10649.713} C_VEL
LIN {X 0,Y 411.202,Z 105.578,A -85,B 0,C 180,E1 -10653.156,E2 -10653.156} C_VEL
LIN {X 0,Y 411.192,Z 105.576,A -85,B 0,C 180,E1 -10656.554,E2 -10656.554} C_VEL
LIN {X 0,Y 411.212,Z 105.571,A -85,B 0,C 180,E1 -10659.729,E2 -10659.729} C_VEL
LIN {X 0,Y 411.174,Z 105.58,A -85,B 0,C 180,E1 -10663.133,E2 -10663.133} C_VEL
LIN {X 0,Y 411.17,Z 105.576,A -85,B 0,C 180,E1 -10665.881,E2 -10665.881} C_VEL
LIN {X 0,Y 411.198,Z 105.58,A -85,B 0,C 180,E1 -10668.766,E2 -10668.766} C_VEL
LIN {X 0,Y 411.194,Z 105.574,A -85,B 0,C 180,E1 -10672.027,E2 -10672.027} C_VEL
LIN {X 0,Y 411.203,Z 105.572,A -85,B 0,C 180,E1 -10675.667,E2 -10675.667} C_VEL
LIN {X 0,Y 411.187,Z 105.576,A -85,B 0,C 180,E1 -10679.153,E2 -10679.153} C_VEL
LIN {X 0,Y 411.257,Z 105.573,A -85,B 0,C 180,E1 -10682.523,E2 -10682.523} C_VEL
LIN {X 0,Y 411.225,Z 105.57,A -85,B 0,C 180,E1 -10685.785,E2 -10685.785} C_VEL
LIN {X 0,Y 411.201,Z 105.574,A -85,B 0,C 180,E1 -10688.967,E2 -10688.967} C_VEL
LIN {X 0,Y 411.252,Z 105.57,A -85,B 0,C 180,E1 -10692.086,E2 -10692.086} C_VEL
LIN {X 0,Y 411.259,Z 105.565,A -85,B 0,C 180,E1 -10695.148,E2 -10695.148} C_VEL
LIN {X 0,Y 411.284,Z 105.568,A -85,B 0,C 180,E1 -10698.168,E2 -10698.168} C_VEL
LIN {X 0,Y 411.482,Z 105.544,A -85,B 0,C 180,E1 -10702.147,E2 -10702.147} C_VEL
LIN {X 0,Y 411.475,Z 105.545,A -85,B 0,C 180,E1 -10704.119,E2 -10704.119} C_VEL
LIN {X 0,Y 411.512,Z 105.54,A -85,B 0,C 180,E1 -10708.043,E2 -10708.043} C_VEL
LIN {X 0,Y 411.641,Z 105.524,A -85,B 0,C 180,E1 -10710.001,E2 -10710.001} C_VEL
LIN {X 0,Y 411.458,Z 105.54,A -85,B 0,C 180,E1 -10712.938,E2 -10712.938} C_VEL
LIN {X 0,Y 411.462,Z 105.54,A -85,B 0,C 180,E1 -10716.868,E2 -10716.868} C_VEL
LIN {X 0,Y 411.294,Z 105.568,A -85,B 0,C 180,E1 -10719.839,E2 -10719.839} C_VEL
LIN {X 0,Y 411.285,Z 105.564,A -85,B 0,C 180,E1 -10723.322,E2 -10723.322} C_VEL
LIN {X 0,Y 411.259,Z 105.565,A -85,B 0,C 180,E1 -10726.889,E2 -10726.889} C_VEL
LIN {X 0,Y 411.242,Z 105.569,A -85,B 0,C 180,E1 -10727.588,E2 -10727.588} C_VEL
LIN {X 0,Y 410.582,Z 105.656,A -85,B 0,C 180,E1 -10728.406,E2 -10728.406} C_VEL
LIN {X 0,Y 407.694,Z 106.018,A -85,B 0,C 180,E1 -10729.734,E2 -10729.734} C_VEL
LIN {X 0,Y 405.25,Z 106.319,A -85,B 0,C 180,E1 -10730.807,E2 -10730.807} C_VEL
LIN {X 0,Y 404.214,Z 106.45,A -85,B 0,C 180,E1 -10731.637,E2 -10731.637} C_VEL
LIN {X 0,Y 404.138,Z 106.452,A -85,B 0,C 180,E1 -10731.918,E2 -10731.918} C_VEL
LIN {X 0,Y 404.218,Z 106.446,A -85,B 0,C 180,E1 -10735.297,E2 -10735.297} C_VEL
LIN {X 0,Y 404.198,Z 106.447,A -85,B 0,C 180,E1 -10738,E2 -10738} C_VEL
LIN {X 0,Y 404.142,Z 106.458,A -85,B 0,C 180,E1 -10741.559,E2 -10741.559} C_VEL
LIN {X 0,Y 404.187,Z 106.449,A -85,B 0,C 180,E1 -10745.017,E2 -10745.017} C_VEL
LIN {X 0,Y 404.158,Z 106.451,A -85,B 0,C 180,E1 -10748.757,E2 -10748.757} C_VEL
LIN {X 0,Y 404.127,Z 106.458,A -85,B 0,C 180,E1 -10751.6,E2 -10751.6} C_VEL
LIN {X 0,Y 404.151,Z 106.451,A -85,B 0,C 180,E1 -10754.523,E2 -10754.523} C_VEL
LIN {X 0,Y 404.139,Z 106.459,A -85,B 0,C 180,E1 -10757.296,E2 -10757.296} C_VEL
LIN {X 0,Y 404.172,Z 106.449,A -85,B 0,C 180,E1 -10759.956,E2 -10759.956} C_VEL
LIN {X 0,Y 404.14,Z 106.459,A -85,B 0,C 180,E1 -10763.125,E2 -10763.125} C_VEL
LIN {X 0,Y 404.148,Z 106.453,A -85,B 0,C 180,E1 -10766.188,E2 -10766.188} C_VEL
LIN {X 0,Y 404.173,Z 106.515,A -85,B 0,C 180,E1 -10766.674,E2 -10766.674} C_VEL
LIN {X 0,Y 405.197,Z 109.322,A -85,B 0,C 180,E1 -10766.826,E2 -10766.826} C_VEL
LIN {X 0,Y 421.828,Z 142.342,A -85,B 0,C 180,E1 -10768.859,E2 -10768.859} C_VEL
LIN {X 0,Y 416.689,Z 296.984,A -85,B 0,C 180,E1 -10772.161,E2 -10772.161} C_VEL
LIN {X 0,Y 416.029,Z 313.323,A -85,B 0,C 180,E1 -10772.693,E2 -10772.693} C_VEL
LIN {X 0,Y 415.083,Z 329.691,A -85,B 0,C 180,E1 -10773.408,E2 -10773.408} C_VEL
LIN {X 0,Y 414.008,Z 345.626,A -85,B 0,C 180,E1 -10774.302,E2 -10774.302} C_VEL
LIN {X 0,Y 412.804,Z 360.785,A -85,B 0,C 180,E1 -10775.347,E2 -10775.347} C_VEL
LIN {X 0,Y 411.423,Z 375.812,A -85,B 0,C 180,E1 -10776.599,E2 -10776.599} C_VEL
LIN {X 0,Y 410.063,Z 389.678,A -85,B 0,C 180,E1 -10777.981,E2 -10777.981} C_VEL
LIN {X 0,Y 408.809,Z 402.451,A -85,B 0,C 180,E1 -10779.496,E2 -10779.496} C_VEL
LIN {X 0,Y 407.572,Z 414.315,A -85,B 0,C 180,E1 -10781.143,E2 -10781.143} C_VEL
LIN {X 0,Y 406.53,Z 425.154,A -85,B 0,C 180,E1 -10782.909,E2 -10782.909} C_VEL
LIN {X 0,Y 405.589,Z 434.465,A -85,B 0,C 180,E1 -10784.678,E2 -10784.678} C_VEL
LIN {X 0,Y 404.846,Z 443.028,A -85,B 0,C 180,E1 -10786.619,E2 -10786.619} C_VEL
LIN {X 0,Y 404.212,Z 449.888,A -85,B 0,C 180,E1 -10788.466,E2 -10788.466} C_VEL
LIN {X 0,Y 403.808,Z 456.123,A -85,B 0,C 180,E1 -10790.483,E2 -10790.483} C_VEL
LIN {X 0,Y 403.536,Z 461.053,A -85,B 0,C 180,E1 -10792.494,E2 -10792.494} C_VEL
LIN {X 0,Y 403.361,Z 464.048,A -85,B 0,C 180,E1 -10793.999,E2 -10793.999} C_VEL
LIN {X 0,Y 403.287,Z 466.986,A -85,B 0,C 180,E1 -10796.003,E2 -10796.003} C_VEL
LIN {X 0,Y 403.2,Z 468.963,A -85,B 0,C 180,E1 -10798.002,E2 -10798.002} C_VEL
LIN {X 0,Y 403.079,Z 469.871,A -85,B 0,C 180,E1 -10800,E2 -10800} C_VEL
LIN {X 0,Y 403.229,Z 469.774,A -85,B 0,C 180,E1 -10801.998,E2 -10801.998} C_VEL
LIN {X 0,Y 403.401,Z 469.367,A -85,B 0,C 180,E1 -10802.996,E2 -10802.996} C_VEL
LIN {X 0,Y 403.482,Z 467.71,A -85,B 0,C 180,E1 -10804.996,E2 -10804.996} C_VEL
LIN {X 0,Y 403.76,Z 464.768,A -85,B 0,C 180,E1 -10807.173,E2 -10807.173} C_VEL
LIN {X 0,Y 404.112,Z 461.324,A -85,B 0,C 180,E1 -10809.005,E2 -10809.005} C_VEL
LIN {X 0,Y 404.682,Z 456.413,A -85,B 0,C 180,E1 -10811.013,E2 -10811.013} C_VEL
LIN {X 0,Y 405.318,Z 450.346,A -85,B 0,C 180,E1 -10813.027,E2 -10813.027} C_VEL
LIN {X 0,Y 406.334,Z 442.87,A -85,B 0,C 180,E1 -10815.037,E2 -10815.037} C_VEL
LIN {X 0,Y 407.561,Z 433.81,A -85,B 0,C 180,E1 -10817.046,E2 -10817.046} C_VEL
LIN {X 0,Y 408.824,Z 424.433,A -85,B 0,C 180,E1 -10818.804,E2 -10818.804} C_VEL
LIN {X 0,Y 410.365,Z 413.436,A -85,B 0,C 180,E1 -10820.554,E2 -10820.554} C_VEL
LIN {X 0,Y 411.795,Z 402.471,A -85,B 0,C 180,E1 -10822.053,E2 -10822.053} C_VEL
LIN {X 0,Y 413.676,Z 388.744,A -85,B 0,C 180,E1 -10823.624,E2 -10823.624} C_VEL
LIN {X 0,Y 415.158,Z 375.62,A -85,B 0,C 180,E1 -10824.904,E2 -10824.904} C_VEL
LIN {X 0,Y 416.871,Z 360.216,A -85,B 0,C 180,E1 -10826.155,E2 -10826.155} C_VEL
LIN {X 0,Y 418.477,Z 344.304,A -85,B 0,C 180,E1 -10827.208,E2 -10827.208} C_VEL
LIN {X 0,Y 419.782,Z 327.812,A -85,B 0,C 180,E1 -10828.091,E2 -10828.091} C_VEL
LIN {X 0,Y 420.937,Z 310.767,A -85,B 0,C 180,E1 -10828.788,E2 -10828.788} C_VEL
LIN {X 0,Y 422.125,Z 289.234,A -85,B 0,C 180,E1 -10829.416,E2 -10829.416} C_VEL
LIN {X 0,Y 426.723,Z 222.699,A -85,B 0,C 180,E1 -10831.196,E2 -10831.196} C_VEL
LIN {X 0,Y 433.205,Z 151.035,A -85,B 0,C 180,E1 -10833.22,E2 -10833.22} C_VEL
LIN {X 0,Y 433.215,Z 149.323,A -85,B 0,C 180,E1 -10833.297,E2 -10833.297} C_VEL
LIN {X 0,Y 428.679,Z 140.813,A -85,B 0,C 180,E1 -10834.525,E2 -10834.525} C_VEL
LIN {X 0,Y 425.206,Z 135.368,A -85,B 0,C 180,E1 -10835.559,E2 -10835.559} C_VEL
LIN {X 0,Y 422.31,Z 131.44,A -85,B 0,C 180,E1 -10836.507,E2 -10836.507} C_VEL
LIN {X 0,Y 417.868,Z 126.065,A -85,B 0,C 180,E1 -10838.258,E2 -10838.258} C_VEL
LIN {X 0,Y 414.075,Z 122.357,A -85,B 0,C 180,E1 -10840.284,E2 -10840.284} C_VEL
LIN {X 0,Y 412.1,Z 120.663,A -85,B 0,C 180,E1 -10841.99,E2 -10841.99} C_VEL
LIN {X 0,Y 411.068,Z 120.431,A -85,B 0,C 180,E1 -10843.823,E2 -10843.823} C_VEL
LIN {X 0,Y 411.745,Z 122.243,A -85,B 0,C 180,E1 -10845.798,E2 -10845.798} C_VEL
LIN {X 0,Y 412.67,Z 123.942,A -85,B 0,C 180,E1 -10847.08,E2 -10847.08} C_VEL
LIN {X 0,Y 414.383,Z 127.672,A -85,B 0,C 180,E1 -10848.945,E2 -10848.945} C_VEL
LIN {X 0,Y 417.377,Z 133.177,A -85,B 0,C 180,E1 -10850.623,E2 -10850.623} C_VEL
LIN {X 0,Y 420.508,Z 138.662,A -85,B 0,C 180,E1 -10851.962,E2 -10851.962} C_VEL
LIN {X 0,Y 424.591,Z 146.65,A -85,B 0,C 180,E1 -10853.433,E2 -10853.433} C_VEL
LIN {X 0,Y 427.599,Z 153.277,A -85,B 0,C 180,E1 -10854.395,E2 -10854.395} C_VEL
LIN {X 0,Y 429.108,Z 157.346,A -85,B 0,C 180,E1 -10854.879,E2 -10854.879} C_VEL
LIN {X 0,Y 430.253,Z 173.039,A -85,B 0,C 180,E1 -10855.796,E2 -10855.796} C_VEL
LIN {X 0,Y 430.985,Z 189.668,A -85,B 0,C 180,E1 -10856.619,E2 -10856.619} C_VEL
LIN {X 0,Y 425.7,Z 254.893,A -85,B 0,C 180,E1 -10858.422,E2 -10858.422} C_VEL
LIN {X 0,Y 421.6,Z 319.815,A -85,B 0,C 180,E1 -10860.135,E2 -10860.135} C_VEL
LIN {X 0,Y 419.648,Z 353.231,A -85,B 0,C 180,E1 -10861.011,E2 -10861.011} C_VEL
LIN {X 0,Y 418.078,Z 371.098,A -85,B 0,C 180,E1 -10861.647,E2 -10861.647} C_VEL
LIN {X 0,Y 416.573,Z 386.443,A -85,B 0,C 180,E1 -10862.357,E2 -10862.357} C_VEL
LIN {X 0,Y 414.718,Z 402.989,A -85,B 0,C 180,E1 -10863.315,E2 -10863.315} C_VEL
LIN {X 0,Y 412.892,Z 418.825,A -85,B 0,C 180,E1 -10864.439,E2 -10864.439} C_VEL
LIN {X 0,Y 411.164,Z 433.096,A -85,B 0,C 180,E1 -10865.646,E2 -10865.646} C_VEL
LIN {X 0,Y 409.378,Z 448.04,A -85,B 0,C 180,E1 -10867.143,E2 -10867.143} C_VEL
LIN {X 0,Y 407.75,Z 461.842,A -85,B 0,C 180,E1 -10868.779,E2 -10868.779} C_VEL
LIN {X 0,Y 406.386,Z 474.558,A -85,B 0,C 180,E1 -10870.554,E2 -10870.554} C_VEL
LIN {X 0,Y 405.183,Z 486.656,A -85,B 0,C 180,E1 -10872.551,E2 -10872.551} C_VEL
LIN {X 0,Y 404.273,Z 497.197,A -85,B 0,C 180,E1 -10874.626,E2 -10874.626} C_VEL
LIN {X 0,Y 403.679,Z 505.839,A -85,B 0,C 180,E1 -10876.662,E2 -10876.662} C_VEL
LIN {X 0,Y 403.284,Z 512.231,A -85,B 0,C 180,E1 -10878.438,E2 -10878.438} C_VEL
LIN {X 0,Y 403.06,Z 518.247,A -85,B 0,C 180,E1 -10880.464,E2 -10880.464} C_VEL
LIN {X 0,Y 403.051,Z 523.011,A -85,B 0,C 180,E1 -10882.485,E2 -10882.485} C_VEL
LIN {X 0,Y 403.081,Z 525.82,A -85,B 0,C 180,E1 -10883.994,E2 -10883.994} C_VEL
LIN {X 0,Y 403.005,Z 528.58,A -85,B 0,C 180,E1 -10885.999,E2 -10885.999} C_VEL
LIN {X 0,Y 403.12,Z 529.563,A -85,B 0,C 180,E1 -10887.001,E2 -10887.001} C_VEL
LIN {X 0,Y 403.098,Z 530.605,A -85,B 0,C 180,E1 -10889,E2 -10889} C_VEL
LIN {X 0,Y 403.097,Z 530.64,A -85,B 0,C 180,E1 -10890.998,E2 -10890.998} C_VEL
LIN {X 0,Y 403.111,Z 529.498,A -85,B 0,C 180,E1 -10892.997,E2 -10892.997} C_VEL
LIN {X 0,Y 403.013,Z 527.297,A -85,B 0,C 180,E1 -10895.001,E2 -10895.001} C_VEL
LIN {X 0,Y 403.129,Z 525.032,A -85,B 0,C 180,E1 -10896.428,E2 -10896.428} C_VEL
LIN {X 0,Y 403.077,Z 520.688,A -85,B 0,C 180,E1 -10898.522,E2 -10898.522} C_VEL
LIN {X 0,Y 403.171,Z 515.16,A -85,B 0,C 180,E1 -10900.546,E2 -10900.546} C_VEL
LIN {X 0,Y 403.532,Z 508.203,A -85,B 0,C 180,E1 -10902.61,E2 -10902.61} C_VEL
LIN {X 0,Y 403.99,Z 500.047,A -85,B 0,C 180,E1 -10904.61,E2 -10904.61} C_VEL
LIN {X 0,Y 404.808,Z 490.079,A -85,B 0,C 180,E1 -10906.645,E2 -10906.645} C_VEL
LIN {X 0,Y 405.658,Z 479.68,A -85,B 0,C 180,E1 -10908.431,E2 -10908.431} C_VEL
LIN {X 0,Y 406.891,Z 467.483,A -85,B 0,C 180,E1 -10910.208,E2 -10910.208} C_VEL
LIN {X 0,Y 408.134,Z 454.99,A -85,B 0,C 180,E1 -10911.757,E2 -10911.757} C_VEL
LIN {X 0,Y 409.571,Z 440.827,A -85,B 0,C 180,E1 -10913.244,E2 -10913.244} C_VEL
LIN {X 0,Y 411.045,Z 426.632,A -85,B 0,C 180,E1 -10914.495,E2 -10914.495} C_VEL
LIN {X 0,Y 412.353,Z 411.873,A -85,B 0,C 180,E1 -10915.584,E2 -10915.584} C_VEL
LIN {X 0,Y 413.794,Z 395.723,A -85,B 0,C 180,E1 -10916.544,E2 -10916.544} C_VEL
LIN {X 0,Y 415.005,Z 379.366,A -85,B 0,C 180,E1 -10917.311,E2 -10917.311} C_VEL
LIN {X 0,Y 416.028,Z 362.96,A -85,B 0,C 180,E1 -10917.886,E2 -10917.886} C_VEL
LIN {X 0,Y 416.835,Z 344.321,A -85,B 0,C 180,E1 -10918.339,E2 -10918.339} C_VEL
LIN {X 0,Y 422.072,Z 187.625,A -85,B 0,C 180,E1 -10921.677,E2 -10921.677} C_VEL
LIN {X 0,Y 416.993,Z 149.14,A -85,B 0,C 180,E1 -10922.997,E2 -10922.997} C_VEL
LIN {X 0,Y 417.131,Z 146.783,A -85,B 0,C 180,E1 -10923.252,E2 -10923.252} C_VEL
LIN {X 0,Y 411.199,Z 127.787,A -85,B 0,C 180,E1 -10925.863,E2 -10925.863} C_VEL
LIN {X 0,Y 404.17,Z 106.454,A -85,B 0,C 180,E1 -10928.998,E2 -10928.998} C_VEL
LIN {X 0,Y 404.202,Z 106.451,A -85,B 0,C 180,E1 -10932.695,E2 -10932.695} C_VEL
LIN {X 0,Y 404.148,Z 106.456,A -85,B 0,C 180,E1 -10935.926,E2 -10935.926} C_VEL
LIN {X 0,Y 404.115,Z 106.459,A -85,B 0,C 180,E1 -10938.635,E2 -10938.635} C_VEL
LIN {X 0,Y 404.154,Z 106.451,A -85,B 0,C 180,E1 -10941.491,E2 -10941.491} C_VEL
LIN {X 0,Y 404.181,Z 106.447,A -85,B 0,C 180,E1 -10944.984,E2 -10944.984} C_VEL
LIN {X 0,Y 404.143,Z 106.455,A -85,B 0,C 180,E1 -10948.554,E2 -10948.554} C_VEL
LIN {X 0,Y 404.193,Z 106.451,A -85,B 0,C 180,E1 -10952,E2 -10952} C_VEL
LIN {X 0,Y 404.172,Z 106.449,A -85,B 0,C 180,E1 -10955.334,E2 -10955.334} C_VEL
LIN {X 0,Y 404.134,Z 106.454,A -85,B 0,C 180,E1 -10958.581,E2 -10958.581} C_VEL
LIN {X 0,Y 404.206,Z 106.449,A -85,B 0,C 180,E1 -10961.762,E2 -10961.762} C_VEL
LIN {X 0,Y 404.208,Z 106.444,A -85,B 0,C 180,E1 -10964.882,E2 -10964.882} C_VEL
LIN {X 0,Y 404.265,Z 106.442,A -85,B 0,C 180,E1 -10967.959,E2 -10967.959} C_VEL
LIN {X 0,Y 404.429,Z 106.419,A -85,B 0,C 180,E1 -10972.1,E2 -10972.1} C_VEL
LIN {X 0,Y 404.419,Z 106.421,A -85,B 0,C 180,E1 -10974.015,E2 -10974.015} C_VEL
LIN {X 0,Y 404.478,Z 106.413,A -85,B 0,C 180,E1 -10978.009,E2 -10978.009} C_VEL
LIN {X 0,Y 404.607,Z 106.397,A -85,B 0,C 180,E1 -10980,E2 -10980} C_VEL
LIN {X 0,Y 404.419,Z 106.419,A -85,B 0,C 180,E1 -10982.989,E2 -10982.989} C_VEL
LIN {X 0,Y 404.407,Z 106.42,A -85,B 0,C 180,E1 -10986.987,E2 -10986.987} C_VEL
LIN {X 0,Y 404.254,Z 106.439,A -85,B 0,C 180,E1 -10990.012,E2 -10990.012} C_VEL
LIN {X 0,Y 404.262,Z 106.442,A -85,B 0,C 180,E1 -10993.212,E2 -10993.212} C_VEL
LIN {X 0,Y 404.211,Z 106.447,A -85,B 0,C 180,E1 -10997.007,E2 -10997.007} C_VEL
LIN {X 0,Y 404.159,Z 106.45,A -85,B 0,C 180,E1 -11000.352,E2 -11000.352} C_VEL
LIN {X 0,Y 404.165,Z 106.452,A -85,B 0,C 180,E1 -11003.575,E2 -11003.575} C_VEL
LIN {X 0,Y 404.179,Z 106.448,A -85,B 0,C 180,E1 -11005.767,E2 -11005.767} C_VEL
LIN {X 0,Y 404.191,Z 106.446,A -85,B 0,C 180,E1 -11008,E2 -11008} C_VEL
LIN {X 0,Y 404.135,Z 106.455,A -85,B 0,C 180,E1 -11011.559,E2 -11011.559} C_VEL
LIN {X 0,Y 404.182,Z 106.454,A -85,B 0,C 180,E1 -11015.016,E2 -11015.016} C_VEL
LIN {X 0,Y 404.154,Z 106.455,A -85,B 0,C 180,E1 -11018.757,E2 -11018.757} C_VEL
LIN {X 0,Y 404.121,Z 106.455,A -85,B 0,C 180,E1 -11021.6,E2 -11021.6} C_VEL
LIN {X 0,Y 404.147,Z 106.454,A -85,B 0,C 180,E1 -11024.523,E2 -11024.523} C_VEL
LIN {X 0,Y 404.17,Z 106.45,A -85,B 0,C 180,E1 -11027.301,E2 -11027.301} C_VEL
LIN {X 0,Y 404.166,Z 106.449,A -85,B 0,C 180,E1 -11029.956,E2 -11029.956} C_VEL
LIN {X 0,Y 404.134,Z 106.455,A -85,B 0,C 180,E1 -11033.126,E2 -11033.126} C_VEL
LIN {X 0,Y 404.142,Z 106.454,A -85,B 0,C 180,E1 -11036.188,E2 -11036.188} C_VEL
LIN {X 0,Y 404.143,Z 106.452,A -85,B 0,C 180,E1 -11039.716,E2 -11039.716} C_VEL
LIN {X 0,Y 404.193,Z 106.447,A -85,B 0,C 180,E1 -11043.124,E2 -11043.124} C_VEL
LIN {X 0,Y 404.175,Z 106.448,A -85,B 0,C 180,E1 -11045.335,E2 -11045.335} C_VEL
LIN {X 0,Y 404.162,Z 106.455,A -85,B 0,C 180,E1 -11048.583,E2 -11048.583} C_VEL
LIN {X 0,Y 404.213,Z 106.444,A -85,B 0,C 180,E1 -11051.763,E2 -11051.763} C_VEL
LIN {X 0,Y 404.206,Z 106.445,A -85,B 0,C 180,E1 -11054.883,E2 -11054.883} C_VEL
LIN {X 0,Y 404.256,Z 106.441,A -85,B 0,C 180,E1 -11057.959,E2 -11057.959} C_VEL
LIN {X 0,Y 404.433,Z 106.422,A -85,B 0,C 180,E1 -11062.1,E2 -11062.1} C_VEL
LIN {X 0,Y 404.424,Z 106.422,A -85,B 0,C 180,E1 -11064.016,E2 -11064.016} C_VEL
LIN {X 0,Y 404.481,Z 106.416,A -85,B 0,C 180,E1 -11068.009,E2 -11068.009} C_VEL
LIN {X 0,Y 404.61,Z 106.4,A -85,B 0,C 180,E1 -11070.001,E2 -11070.001} C_VEL
LIN {X 0,Y 404.417,Z 106.418,A -85,B 0,C 180,E1 -11072.989,E2 -11072.989} C_VEL
LIN {X 0,Y 404.413,Z 106.418,A -85,B 0,C 180,E1 -11076.988,E2 -11076.988} C_VEL
LIN {X 0,Y 404.26,Z 106.443,A -85,B 0,C 180,E1 -11080.012,E2 -11080.012} C_VEL
LIN {X 0,Y 404.268,Z 106.437,A -85,B 0,C 180,E1 -11083.212,E2 -11083.212} C_VEL
LIN {X 0,Y 404.218,Z 106.443,A -85,B 0,C 180,E1 -11087.008,E2 -11087.008} C_VEL
LIN {X 0,Y 404.166,Z 106.45,A -85,B 0,C 180,E1 -11090.352,E2 -11090.352} C_VEL
LIN {X 0,Y 404.138,Z 106.452,A -85,B 0,C 180,E1 -11091.918,E2 -11091.918} C_VEL
LIN {X 0,Y 403.495,Z 106.533,A -85,B 0,C 180,E1 -11092.75,E2 -11092.75} C_VEL
LIN {X 0,Y 400.663,Z 106.887,A -85,B 0,C 180,E1 -11094.102,E2 -11094.102} C_VEL
LIN {X 0,Y 398.253,Z 107.188,A -85,B 0,C 180,E1 -11095.194,E2 -11095.194} C_VEL
LIN {X 0,Y 397.219,Z 107.317,A -85,B 0,C 180,E1 -11096.038,E2 -11096.038} C_VEL
LIN {X 0,Y 397.136,Z 107.325,A -85,B 0,C 180,E1 -11096.324,E2 -11096.324} C_VEL
LIN {X 0,Y 397.124,Z 107.326,A -85,B 0,C 180,E1 -11098.544,E2 -11098.544} C_VEL
LIN {X 0,Y 397.081,Z 107.333,A -85,B 0,C 180,E1 -11102.072,E2 -11102.072} C_VEL
LIN {X 0,Y 397.122,Z 107.333,A -85,B 0,C 180,E1 -11105.504,E2 -11105.504} C_VEL
LIN {X 0,Y 397.133,Z 107.327,A -85,B 0,C 180,E1 -11108.862,E2 -11108.862} C_VEL
LIN {X 0,Y 397.073,Z 107.332,A -85,B 0,C 180,E1 -11112.267,E2 -11112.267} C_VEL
LIN {X 0,Y 397.092,Z 107.335,A -85,B 0,C 180,E1 -11115.069,E2 -11115.069} C_VEL
LIN {X 0,Y 397.069,Z 107.333,A -85,B 0,C 180,E1 -11118.022,E2 -11118.022} C_VEL
LIN {X 0,Y 397.131,Z 107.332,A -85,B 0,C 180,E1 -11121.139,E2 -11121.139} C_VEL
LIN {X 0,Y 397.123,Z 107.331,A -85,B 0,C 180,E1 -11124.497,E2 -11124.497} C_VEL
LIN {X 0,Y 397.141,Z 107.529,A -85,B 0,C 180,E1 -11126.155,E2 -11126.155} C_VEL
LIN {X 0,Y 398.217,Z 110.337,A -85,B 0,C 180,E1 -11126.314,E2 -11126.314} C_VEL
LIN {X 0,Y 415.274,Z 144.186,A -85,B 0,C 180,E1 -11128.448,E2 -11128.448} C_VEL
LIN {X 0,Y 415.01,Z 155.986,A -85,B 0,C 180,E1 -11128.718,E2 -11128.718} C_VEL
LIN {X 0,Y 410.076,Z 297.631,A -85,B 0,C 180,E1 -11131.811,E2 -11131.811} C_VEL
LIN {X 0,Y 409.407,Z 313.858,A -85,B 0,C 180,E1 -11132.353,E2 -11132.353} C_VEL
LIN {X 0,Y 408.426,Z 330.165,A -85,B 0,C 180,E1 -11133.078,E2 -11133.078} C_VEL
LIN {X 0,Y 407.299,Z 346.392,A -85,B 0,C 180,E1 -11134.005,E2 -11134.005} C_VEL
LIN {X 0,Y 405.912,Z 362.853,A -85,B 0,C 180,E1 -11135.174,E2 -11135.174} C_VEL
LIN {X 0,Y 404.482,Z 377.609,A -85,B 0,C 180,E1 -11136.445,E2 -11136.445} C_VEL
LIN {X 0,Y 403.121,Z 391.304,A -85,B 0,C 180,E1 -11137.851,E2 -11137.851} C_VEL
LIN {X 0,Y 401.929,Z 402.968,A -85,B 0,C 180,E1 -11139.263,E2 -11139.263} C_VEL
LIN {X 0,Y 400.717,Z 413.966,A -85,B 0,C 180,E1 -11140.801,E2 -11140.801} C_VEL
LIN {X 0,Y 399.665,Z 424.997,A -85,B 0,C 180,E1 -11142.606,E2 -11142.606} C_VEL
LIN {X 0,Y 398.64,Z 434.406,A -85,B 0,C 180,E1 -11144.404,E2 -11144.404} C_VEL
LIN {X 0,Y 397.896,Z 442.67,A -85,B 0,C 180,E1 -11146.28,E2 -11146.28} C_VEL
LIN {X 0,Y 397.211,Z 450.05,A -85,B 0,C 180,E1 -11148.26,E2 -11148.26} C_VEL
LIN {X 0,Y 396.757,Z 456.382,A -85,B 0,C 180,E1 -11150.312,E2 -11150.312} C_VEL
LIN {X 0,Y 396.492,Z 461.376,A -85,B 0,C 180,E1 -11152.36,E2 -11152.36} C_VEL
LIN {X 0,Y 396.297,Z 464.415,A -85,B 0,C 180,E1 -11153.892,E2 -11153.892} C_VEL
LIN {X 0,Y 396.213,Z 467.434,A -85,B 0,C 180,E1 -11155.931,E2 -11155.931} C_VEL
LIN {X 0,Y 396.122,Z 469.481,A -85,B 0,C 180,E1 -11157.966,E2 -11157.966} C_VEL
LIN {X 0,Y 396.025,Z 470.427,A -85,B 0,C 180,E1 -11160,E2 -11160} C_VEL
LIN {X 0,Y 396.184,Z 470.394,A -85,B 0,C 180,E1 -11162.033,E2 -11162.033} C_VEL
LIN {X 0,Y 396.357,Z 470.006,A -85,B 0,C 180,E1 -11163.049,E2 -11163.049} C_VEL
LIN {X 0,Y 396.445,Z 468.397,A -85,B 0,C 180,E1 -11165.085,E2 -11165.085} C_VEL
LIN {X 0,Y 396.724,Z 465.638,A -85,B 0,C 180,E1 -11167.229,E2 -11167.229} C_VEL
LIN {X 0,Y 397.144,Z 462.104,A -85,B 0,C 180,E1 -11169.164,E2 -11169.164} C_VEL
LIN {X 0,Y 397.751,Z 457.258,A -85,B 0,C 180,E1 -11171.207,E2 -11171.207} C_VEL
LIN {X 0,Y 398.435,Z 451.256,A -85,B 0,C 180,E1 -11173.256,E2 -11173.256} C_VEL
LIN {X 0,Y 399.529,Z 443.824,A -85,B 0,C 180,E1 -11175.299,E2 -11175.299} C_VEL
LIN {X 0,Y 400.824,Z 434.853,A -85,B 0,C 180,E1 -11177.342,E2 -11177.342} C_VEL
LIN {X 0,Y 402.199,Z 425.568,A -85,B 0,C 180,E1 -11179.126,E2 -11179.126} C_VEL
LIN {X 0,Y 403.825,Z 414.689,A -85,B 0,C 180,E1 -11180.902,E2 -11180.902} C_VEL
LIN {X 0,Y 405.342,Z 403.827,A -85,B 0,C 180,E1 -11182.423,E2 -11182.423} C_VEL
LIN {X 0,Y 407.255,Z 391.056,A -85,B 0,C 180,E1 -11183.924,E2 -11183.924} C_VEL
LIN {X 0,Y 408.924,Z 377.376,A -85,B 0,C 180,E1 -11185.31,E2 -11185.31} C_VEL
LIN {X 0,Y 410.753,Z 362.08,A -85,B 0,C 180,E1 -11186.594,E2 -11186.594} C_VEL
LIN {X 0,Y 412.539,Z 345.763,A -85,B 0,C 180,E1 -11187.708,E2 -11187.708} C_VEL
LIN {X 0,Y 414.035,Z 328.557,A -85,B 0,C 180,E1 -11188.654,E2 -11188.654} C_VEL
LIN {X 0,Y 415.342,Z 310.981,A -85,B 0,C 180,E1 -11189.387,E2 -11189.387} C_VEL
LIN {X 0,Y 416.69,Z 288.851,A -85,B 0,C 180,E1 -11190.047,E2 -11190.047} C_VEL
LIN {X 0,Y 421.729,Z 223.01,A -85,B 0,C 180,E1 -11191.874,E2 -11191.874} C_VEL
LIN {X 0,Y 428.642,Z 152.959,A -85,B 0,C 180,E1 -11193.919,E2 -11193.919} C_VEL
LIN {X 0,Y 425.065,Z 145.918,A -85,B 0,C 180,E1 -11194.982,E2 -11194.982} C_VEL
LIN {X 0,Y 421.988,Z 141.038,A -85,B 0,C 180,E1 -11195.96,E2 -11195.96} C_VEL
LIN {X 0,Y 419.342,Z 137.432,A -85,B 0,C 180,E1 -11196.888,E2 -11196.888} C_VEL
LIN {X 0,Y 415.464,Z 132.496,A -85,B 0,C 180,E1 -11198.519,E2 -11198.519} C_VEL
LIN {X 0,Y 411.817,Z 128.754,A -85,B 0,C 180,E1 -11200.645,E2 -11200.645} C_VEL
LIN {X 0,Y 409.949,Z 127.327,A -85,B 0,C 180,E1 -11202.508,E2 -11202.508} C_VEL
LIN {X 0,Y 409.261,Z 127.523,A -85,B 0,C 180,E1 -11204.112,E2 -11204.112} C_VEL
LIN {X 0,Y 409.598,Z 129.42,A -85,B 0,C 180,E1 -11206.108,E2 -11206.108} C_VEL
LIN {X 0,Y 410.792,Z 131.672,A -85,B 0,C 180,E1 -11207.575,E2 -11207.575} C_VEL
LIN {X 0,Y 412.555,Z 134.926,A -85,B 0,C 180,E1 -11208.961,E2 -11208.961} C_VEL
LIN {X 0,Y 415.589,Z 140.76,A -85,B 0,C 180,E1 -11210.679,E2 -11210.679} C_VEL
LIN {X 0,Y 417.813,Z 144.995,A -85,B 0,C 180,E1 -11211.677,E2 -11211.677} C_VEL
LIN {X 0,Y 421.386,Z 152.351,A -85,B 0,C 180,E1 -11213.056,E2 -11213.056} C_VEL
LIN {X 0,Y 424.078,Z 158.749,A -85,B 0,C 180,E1 -11213.992,E2 -11213.992} C_VEL
LIN {X 0,Y 424.901,Z 161.282,A -85,B 0,C 180,E1 -11214.292,E2 -11214.292} C_VEL
LIN {X 0,Y 425.693,Z 175.499,A -85,B 0,C 180,E1 -11215.145,E2 -11215.145} C_VEL
LIN {X 0,Y 426.184,Z 191.289,A -85,B 0,C 180,E1 -11215.952,E2 -11215.952} C_VEL
LIN {X 0,Y 419.953,Z 262.349,A -85,B 0,C 180,E1 -11217.974,E2 -11217.974} C_VEL
LIN {X 0,Y 415.377,Z 329.535,A -85,B 0,C 180,E1 -11219.788,E2 -11219.788} C_VEL
LIN {X 0,Y 413.768,Z 354.382,A -85,B 0,C 180,E1 -11220.489,E2 -11220.489} C_VEL
LIN {X 0,Y 411.904,Z 372.851,A -85,B 0,C 180,E1 -11221.183,E2 -11221.183} C_VEL
LIN {X 0,Y 410.24,Z 388.562,A -85,B 0,C 180,E1 -11221.962,E2 -11221.962} C_VEL
LIN {X 0,Y 408.204,Z 405.419,A -85,B 0,C 180,E1 -11222.993,E2 -11222.993} C_VEL
LIN {X 0,Y 406.205,Z 421.155,A -85,B 0,C 180,E1 -11224.164,E2 -11224.164} C_VEL
LIN {X 0,Y 404.344,Z 435.867,A -85,B 0,C 180,E1 -11225.481,E2 -11225.481} C_VEL
LIN {X 0,Y 402.476,Z 450.21,A -85,B 0,C 180,E1 -11227.001,E2 -11227.001} C_VEL
LIN {X 0,Y 400.798,Z 463.534,A -85,B 0,C 180,E1 -11228.662,E2 -11228.662} C_VEL
LIN {X 0,Y 399.386,Z 475.857,A -85,B 0,C 180,E1 -11230.467,E2 -11230.467} C_VEL
LIN {X 0,Y 398.185,Z 487.032,A -85,B 0,C 180,E1 -11232.383,E2 -11232.383} C_VEL
LIN {X 0,Y 397.313,Z 496.796,A -85,B 0,C 180,E1 -11234.35,E2 -11234.35} C_VEL
LIN {X 0,Y 396.665,Z 505.399,A -85,B 0,C 180,E1 -11236.422,E2 -11236.422} C_VEL
LIN {X 0,Y 396.24,Z 511.756,A -85,B 0,C 180,E1 -11238.23,E2 -11238.23} C_VEL
LIN {X 0,Y 395.971,Z 517.771,A -85,B 0,C 180,E1 -11240.292,E2 -11240.292} C_VEL
LIN {X 0,Y 395.977,Z 522.51,A -85,B 0,C 180,E1 -11242.35,E2 -11242.35} C_VEL
LIN {X 0,Y 396.001,Z 525.312,A -85,B 0,C 180,E1 -11243.887,E2 -11243.887} C_VEL
LIN {X 0,Y 395.918,Z 528.045,A -85,B 0,C 180,E1 -11245.928,E2 -11245.928} C_VEL
LIN {X 0,Y 396.05,Z 529.03,A -85,B 0,C 180,E1 -11246.948,E2 -11246.948} C_VEL
LIN {X 0,Y 396.046,Z 530.048,A -85,B 0,C 180,E1 -11248.983,E2 -11248.983} C_VEL
LIN {X 0,Y 396.045,Z 530.044,A -85,B 0,C 180,E1 -11251.016,E2 -11251.016} C_VEL
LIN {X 0,Y 396.043,Z 528.884,A -85,B 0,C 180,E1 -11253.051,E2 -11253.051} C_VEL
LIN {X 0,Y 395.952,Z 526.63,A -85,B 0,C 180,E1 -11255.091,E2 -11255.091} C_VEL
LIN {X 0,Y 395.988,Z 523.253,A -85,B 0,C 180,E1 -11257.136,E2 -11257.136} C_VEL
LIN {X 0,Y 395.98,Z 518.614,A -85,B 0,C 180,E1 -11259.191,E2 -11259.191} C_VEL
LIN {X 0,Y 396.197,Z 512.763,A -85,B 0,C 180,E1 -11261.251,E2 -11261.251} C_VEL
LIN {X 0,Y 396.614,Z 505.526,A -85,B 0,C 180,E1 -11263.318,E2 -11263.318} C_VEL
LIN {X 0,Y 397.189,Z 496.682,A -85,B 0,C 180,E1 -11265.391,E2 -11265.391} C_VEL
LIN {X 0,Y 397.934,Z 487.508,A -85,B 0,C 180,E1 -11267.206,E2 -11267.206} C_VEL
LIN {X 0,Y 398.902,Z 476.785,A -85,B 0,C 180,E1 -11269.022,E2 -11269.022} C_VEL
LIN {X 0,Y 400.072,Z 466.102,A -85,B 0,C 180,E1 -11270.568,E2 -11270.568} C_VEL
LIN {X 0,Y 401.332,Z 453.652,A -85,B 0,C 180,E1 -11272.116,E2 -11272.116} C_VEL
LIN {X 0,Y 402.846,Z 439.01,A -85,B 0,C 180,E1 -11273.656,E2 -11273.656} C_VEL
LIN {X 0,Y 404.506,Z 423.267,A -85,B 0,C 180,E1 -11275.026,E2 -11275.026} C_VEL
LIN {X 0,Y 405.887,Z 408.91,A -85,B 0,C 180,E1 -11276.063,E2 -11276.063} C_VEL
LIN {X 0,Y 407.289,Z 392.989,A -85,B 0,C 180,E1 -11277.002,E2 -11277.002} C_VEL
LIN {X 0,Y 408.621,Z 375.282,A -85,B 0,C 180,E1 -11277.809,E2 -11277.809} C_VEL
LIN {X 0,Y 409.762,Z 357.588,A -85,B 0,C 180,E1 -11278.386,E2 -11278.386} C_VEL
LIN {X 0,Y 415.655,Z 188.231,A -85,B 0,C 180,E1 -11282.103,E2 -11282.103} C_VEL
LIN {X 0,Y 410.45,Z 148.746,A -85,B 0,C 180,E1 -11283.494,E2 -11283.494} C_VEL
LIN {X 0,Y 404.34,Z 129.18,A -85,B 0,C 180,E1 -11286.225,E2 -11286.225} C_VEL
LIN {X 0,Y 398.047,Z 110.342,A -85,B 0,C 180,E1 -11289.025,E2 -11289.025} C_VEL
LIN {X 0,Y 397.137,Z 107.33,A -85,B 0,C 180,E1 -11289.5,E2 -11289.5} C_VEL
LIN {X 0,Y 397.153,Z 107.329,A -85,B 0,C 180,E1 -11292.255,E2 -11292.255} C_VEL
LIN {X 0,Y 397.106,Z 107.333,A -85,B 0,C 180,E1 -11295.065,E2 -11295.065} C_VEL
LIN {X 0,Y 397.063,Z 107.337,A -85,B 0,C 180,E1 -11298.021,E2 -11298.021} C_VEL
LIN {X 0,Y 397.129,Z 107.326,A -85,B 0,C 180,E1 -11301.138,E2 -11301.138} C_VEL
LIN {X 0,Y 397.115,Z 107.331,A -85,B 0,C 180,E1 -11304.496,E2 -11304.496} C_VEL
LIN {X 0,Y 397.106,Z 107.332,A -85,B 0,C 180,E1 -11307.931,E2 -11307.931} C_VEL
LIN {X 0,Y 397.121,Z 107.327,A -85,B 0,C 180,E1 -11311.457,E2 -11311.457} C_VEL
LIN {X 0,Y 397.148,Z 107.326,A -85,B 0,C 180,E1 -11314.487,E2 -11314.487} C_VEL
LIN {X 0,Y 397.104,Z 107.329,A -85,B 0,C 180,E1 -11317.086,E2 -11317.086} C_VEL
LIN {X 0,Y 397.143,Z 107.326,A -85,B 0,C 180,E1 -11320.353,E2 -11320.353} C_VEL
LIN {X 0,Y 397.166,Z 107.324,A -85,B 0,C 180,E1 -11323.553,E2 -11323.553} C_VEL
LIN {X 0,Y 397.224,Z 107.314,A -85,B 0,C 180,E1 -11326.703,E2 -11326.703} C_VEL
LIN {X 0,Y 397.224,Z 107.321,A -85,B 0,C 180,E1 -11329.809,E2 -11329.809} C_VEL
LIN {X 0,Y 397.359,Z 107.297,A -85,B 0,C 180,E1 -11332.888,E2 -11332.888} C_VEL
LIN {X 0,Y 397.251,Z 107.311,A -85,B 0,C 180,E1 -11334.925,E2 -11334.925} C_VEL
LIN {X 0,Y 397.447,Z 107.289,A -85,B 0,C 180,E1 -11337.973,E2 -11337.973} C_VEL
LIN {X 0,Y 397.576,Z 107.273,A -85,B 0,C 180,E1 -11340,E2 -11340} C_VEL
LIN {X 0,Y 397.377,Z 107.296,A -85,B 0,C 180,E1 -11343.042,E2 -11343.042} C_VEL
LIN {X 0,Y 397.36,Z 107.299,A -85,B 0,C 180,E1 -11347.112,E2 -11347.112} C_VEL
LIN {X 0,Y 397.213,Z 107.315,A -85,B 0,C 180,E1 -11350.191,E2 -11350.191} C_VEL
LIN {X 0,Y 397.222,Z 107.32,A -85,B 0,C 180,E1 -11353.321,E2 -11353.321} C_VEL
LIN {X 0,Y 397.177,Z 107.324,A -85,B 0,C 180,E1 -11357.155,E2 -11357.155} C_VEL
LIN {X 0,Y 397.098,Z 107.331,A -85,B 0,C 180,E1 -11360.73,E2 -11360.73} C_VEL
LIN {X 0,Y 397.129,Z 107.326,A -85,B 0,C 180,E1 -11364.019,E2 -11364.019} C_VEL
LIN {X 0,Y 397.19,Z 107.322,A -85,B 0,C 180,E1 -11367.39,E2 -11367.39} C_VEL
LIN {X 0,Y 397.075,Z 107.337,A -85,B 0,C 180,E1 -11370.883,E2 -11370.883} C_VEL
LIN {X 0,Y 397.122,Z 107.328,A -85,B 0,C 180,E1 -11374.494,E2 -11374.494} C_VEL
LIN {X 0,Y 397.102,Z 107.329,A -85,B 0,C 180,E1 -11378.275,E2 -11378.275} C_VEL
LIN {X 0,Y 397.085,Z 107.338,A -85,B 0,C 180,E1 -11380.909,E2 -11380.909} C_VEL
LIN {X 0,Y 397.1,Z 107.329,A -85,B 0,C 180,E1 -11383.649,E2 -11383.649} C_VEL
LIN {X 0,Y 397.104,Z 107.332,A -85,B 0,C 180,E1 -11386.521,E2 -11386.521} C_VEL
LIN {X 0,Y 397.116,Z 107.327,A -85,B 0,C 180,E1 -11389.552,E2 -11389.552} C_VEL
LIN {X 0,Y 397.092,Z 107.336,A -85,B 0,C 180,E1 -11392.791,E2 -11392.791} C_VEL
LIN {X 0,Y 397.116,Z 107.33,A -85,B 0,C 180,E1 -11396.283,E2 -11396.283} C_VEL
LIN {X 0,Y 397.103,Z 107.331,A -85,B 0,C 180,E1 -11400.136,E2 -11400.136} C_VEL
LIN {X 0,Y 397.192,Z 107.324,A -85,B 0,C 180,E1 -11402.611,E2 -11402.611} C_VEL
LIN {X 0,Y 397.131,Z 107.327,A -85,B 0,C 180,E1 -11405.982,E2 -11405.982} C_VEL
LIN {X 0,Y 397.153,Z 107.323,A -85,B 0,C 180,E1 -11409.699,E2 -11409.699} C_VEL
LIN {X 0,Y 397.181,Z 107.321,A -85,B 0,C 180,E1 -11412.846,E2 -11412.846} C_VEL
LIN {X 0,Y 397.228,Z 107.316,A -85,B 0,C 180,E1 -11416.703,E2 -11416.703} C_VEL
LIN {X 0,Y 397.224,Z 107.316,A -85,B 0,C 180,E1 -11419.81,E2 -11419.81} C_VEL
LIN {X 0,Y 397.364,Z 107.297,A -85,B 0,C 180,E1 -11422.889,E2 -11422.889} C_VEL
LIN {X 0,Y 397.255,Z 107.31,A -85,B 0,C 180,E1 -11424.926,E2 -11424.926} C_VEL
LIN {X 0,Y 397.45,Z 107.291,A -85,B 0,C 180,E1 -11427.974,E2 -11427.974} C_VEL
LIN {X 0,Y 397.579,Z 107.276,A -85,B 0,C 180,E1 -11430.001,E2 -11430.001} C_VEL
LIN {X 0,Y 397.376,Z 107.295,A -85,B 0,C 180,E1 -11433.042,E2 -11433.042} C_VEL
LIN {X 0,Y 397.365,Z 107.296,A -85,B 0,C 180,E1 -11437.112,E2 -11437.112} C_VEL
LIN {X 0,Y 397.219,Z 107.318,A -85,B 0,C 180,E1 -11440.192,E2 -11440.192} C_VEL
LIN {X 0,Y 397.228,Z 107.315,A -85,B 0,C 180,E1 -11443.322,E2 -11443.322} C_VEL
LIN {X 0,Y 397.184,Z 107.32,A -85,B 0,C 180,E1 -11447.156,E2 -11447.156} C_VEL
LIN {X 0,Y 397.105,Z 107.328,A -85,B 0,C 180,E1 -11450.73,E2 -11450.73} C_VEL
LIN {X 0,Y 397.134,Z 107.328,A -85,B 0,C 180,E1 -11454.019,E2 -11454.019} C_VEL
LIN {X 0,Y 397.136,Z 107.325,A -85,B 0,C 180,E1 -11456.324,E2 -11456.324} C_VEL
LIN {X 0,Y 396.466,Z 107.412,A -85,B 0,C 180,E1 -11457.171,E2 -11457.171} C_VEL
LIN {X 0,Y 393.592,Z 107.766,A -85,B 0,C 180,E1 -11458.546,E2 -11458.546} C_VEL
LIN {X 0,Y 391.154,Z 108.075,A -85,B 0,C 180,E1 -11459.658,E2 -11459.658} C_VEL
LIN {X 0,Y 390.102,Z 108.201,A -85,B 0,C 180,E1 -11460.517,E2 -11460.517} C_VEL
LIN {X 0,Y 390.014,Z 108.212,A -85,B 0,C 180,E1 -11460.809,E2 -11460.809} C_VEL
LIN {X 0,Y 390.071,Z 108.206,A -85,B 0,C 180,E1 -11464.025,E2 -11464.025} C_VEL
LIN {X 0,Y 390.046,Z 108.213,A -85,B 0,C 180,E1 -11467.551,E2 -11467.551} C_VEL
LIN {X 0,Y 390.06,Z 108.208,A -85,B 0,C 180,E1 -11470.822,E2 -11470.822} C_VEL
LIN {X 0,Y 390.06,Z 108.207,A -85,B 0,C 180,E1 -11473.887,E2 -11473.887} C_VEL
LIN {X 0,Y 390.06,Z 108.208,A -85,B 0,C 180,E1 -11476.79,E2 -11476.79} C_VEL
LIN {X 0,Y 390.059,Z 108.209,A -85,B 0,C 180,E1 -11479.561,E2 -11479.561} C_VEL
LIN {X 0,Y 390.046,Z 108.208,A -85,B 0,C 180,E1 -11482.45,E2 -11482.45} C_VEL
LIN {X 0,Y 390.094,Z 108.303,A -85,B 0,C 180,E1 -11485.609,E2 -11485.609} C_VEL
LIN {X 0,Y 391.156,Z 111.143,A -85,B 0,C 180,E1 -11485.774,E2 -11485.774} C_VEL
LIN {X 0,Y 408.444,Z 145.412,A -85,B 0,C 180,E1 -11487.994,E2 -11487.994} C_VEL
LIN {X 0,Y 408.935,Z 146.395,A -85,B 0,C 180,E1 -11488.054,E2 -11488.054} C_VEL
LIN {X 0,Y 403.985,Z 283.213,A -85,B 0,C 180,E1 -11491.099,E2 -11491.099} C_VEL
LIN {X 0,Y 403.207,Z 303.155,A -85,B 0,C 180,E1 -11491.607,E2 -11491.607} C_VEL
LIN {X 0,Y 402.371,Z 320.307,A -85,B 0,C 180,E1 -11492.251,E2 -11492.251} C_VEL
LIN {X 0,Y 401.28,Z 337.299,A -85,B 0,C 180,E1 -11493.103,E2 -11493.103} C_VEL
LIN {X 0,Y 400.103,Z 352.91,A -85,B 0,C 180,E1 -11494.091,E2 -11494.091} C_VEL
LIN {X 0,Y 398.71,Z 368.009,A -85,B 0,C 180,E1 -11495.251,E2 -11495.251} C_VEL
LIN {X 0,Y 397.216,Z 383.305,A -85,B 0,C 180,E1 -11496.679,E2 -11496.679} C_VEL
LIN {X 0,Y 395.708,Z 397.249,A -85,B 0,C 180,E1 -11498.238,E2 -11498.238} C_VEL
LIN {X 0,Y 394.294,Z 410.033,A -85,B 0,C 180,E1 -11499.933,E2 -11499.933} C_VEL
LIN {X 0,Y 393.089,Z 421.882,A -85,B 0,C 180,E1 -11501.793,E2 -11501.793} C_VEL
LIN {X 0,Y 392.026,Z 431.692,A -85,B 0,C 180,E1 -11503.599,E2 -11503.599} C_VEL
LIN {X 0,Y 391.148,Z 440.237,A -85,B 0,C 180,E1 -11505.431,E2 -11505.431} C_VEL
LIN {X 0,Y 390.399,Z 448.369,A -85,B 0,C 180,E1 -11507.524,E2 -11507.524} C_VEL
LIN {X 0,Y 389.822,Z 455.072,A -85,B 0,C 180,E1 -11509.613,E2 -11509.613} C_VEL
LIN {X 0,Y 389.473,Z 460.528,A -85,B 0,C 180,E1 -11511.7,E2 -11511.7} C_VEL
LIN {X 0,Y 389.239,Z 464.766,A -85,B 0,C 180,E1 -11513.781,E2 -11513.781} C_VEL
LIN {X 0,Y 389.126,Z 467.872,A -85,B 0,C 180,E1 -11515.857,E2 -11515.857} C_VEL
LIN {X 0,Y 389.047,Z 469.986,A -85,B 0,C 180,E1 -11517.929,E2 -11517.929} C_VEL
LIN {X 0,Y 388.973,Z 470.983,A -85,B 0,C 180,E1 -11520,E2 -11520} C_VEL
LIN {X 0,Y 389.14,Z 471.022,A -85,B 0,C 180,E1 -11522.07,E2 -11522.07} C_VEL
LIN {X 0,Y 389.314,Z 470.644,A -85,B 0,C 180,E1 -11523.104,E2 -11523.104} C_VEL
LIN {X 0,Y 389.409,Z 469.098,A -85,B 0,C 180,E1 -11525.177,E2 -11525.177} C_VEL
LIN {X 0,Y 389.706,Z 466.496,A -85,B 0,C 180,E1 -11527.305,E2 -11527.305} C_VEL
LIN {X 0,Y 390.303,Z 461.856,A -85,B 0,C 180,E1 -11529.849,E2 -11529.849} C_VEL
LIN {X 0,Y 391.032,Z 456.762,A -85,B 0,C 180,E1 -11531.928,E2 -11531.928} C_VEL
LIN {X 0,Y 391.842,Z 450.455,A -85,B 0,C 180,E1 -11534.012,E2 -11534.012} C_VEL
LIN {X 0,Y 393.045,Z 442.767,A -85,B 0,C 180,E1 -11536.09,E2 -11536.09} C_VEL
LIN {X 0,Y 394.5,Z 433.514,A -85,B 0,C 180,E1 -11538.165,E2 -11538.165} C_VEL
LIN {X 0,Y 396.043,Z 424.039,A -85,B 0,C 180,E1 -11539.947,E2 -11539.947} C_VEL
LIN {X 0,Y 397.847,Z 412.597,A -85,B 0,C 180,E1 -11541.775,E2 -11541.775} C_VEL
LIN {X 0,Y 399.687,Z 400.323,A -85,B 0,C 180,E1 -11543.438,E2 -11543.438} C_VEL
LIN {X 0,Y 401.739,Z 386.893,A -85,B 0,C 180,E1 -11544.963,E2 -11544.963} C_VEL
LIN {X 0,Y 403.537,Z 373.835,A -85,B 0,C 180,E1 -11546.227,E2 -11546.227} C_VEL
LIN {X 0,Y 405.364,Z 359.173,A -85,B 0,C 180,E1 -11547.423,E2 -11547.423} C_VEL
LIN {X 0,Y 407.164,Z 343.317,A -85,B 0,C 180,E1 -11548.478,E2 -11548.478} C_VEL
LIN {X 0,Y 408.621,Z 327.185,A -85,B 0,C 180,E1 -11549.352,E2 -11549.352} C_VEL
LIN {X 0,Y 410.003,Z 309.342,A -85,B 0,C 180,E1 -11550.091,E2 -11550.091} C_VEL
LIN {X 0,Y 412.444,Z 275.382,A -85,B 0,C 180,E1 -11551.076,E2 -11551.076} C_VEL
LIN {X 0,Y 418.244,Z 209.819,A -85,B 0,C 180,E1 -11552.993,E2 -11552.993} C_VEL
LIN {X 0,Y 424.08,Z 156.154,A -85,B 0,C 180,E1 -11554.622,E2 -11554.622} C_VEL
LIN {X 0,Y 420.735,Z 149.635,A -85,B 0,C 180,E1 -11555.723,E2 -11555.723} C_VEL
LIN {X 0,Y 417.149,Z 144.206,A -85,B 0,C 180,E1 -11557.005,E2 -11557.005} C_VEL
LIN {X 0,Y 413.299,Z 139.143,A -85,B 0,C 180,E1 -11558.691,E2 -11558.691} C_VEL
LIN {X 0,Y 409.832,Z 135.507,A -85,B 0,C 180,E1 -11560.809,E2 -11560.809} C_VEL
LIN {X 0,Y 408.374,Z 134.284,A -85,B 0,C 180,E1 -11562.266,E2 -11562.266} C_VEL
LIN {X 0,Y 407.537,Z 134.346,A -85,B 0,C 180,E1 -11563.997,E2 -11563.997} C_VEL
LIN {X 0,Y 407.716,Z 136.074,A -85,B 0,C 180,E1 -11565.862,E2 -11565.862} C_VEL
LIN {X 0,Y 408.769,Z 138.268,A -85,B 0,C 180,E1 -11567.339,E2 -11567.339} C_VEL
LIN {X 0,Y 410.315,Z 141.32,A -85,B 0,C 180,E1 -11568.673,E2 -11568.673} C_VEL
LIN {X 0,Y 413.419,Z 147.69,A -85,B 0,C 180,E1 -11570.56,E2 -11570.56} C_VEL
LIN {X 0,Y 415.596,Z 152.284,A -85,B 0,C 180,E1 -11571.59,E2 -11571.59} C_VEL
LIN {X 0,Y 418.105,Z 157.853,A -85,B 0,C 180,E1 -11572.626,E2 -11572.626} C_VEL
LIN {X 0,Y 420.407,Z 163.655,A -85,B 0,C 180,E1 -11573.505,E2 -11573.505} C_VEL
LIN {X 0,Y 420.835,Z 165.498,A -85,B 0,C 180,E1 -11573.7,E2 -11573.7} C_VEL
LIN {X 0,Y 421.312,Z 177.804,A -85,B 0,C 180,E1 -11574.456,E2 -11574.456} C_VEL
LIN {X 0,Y 421.567,Z 192.304,A -85,B 0,C 180,E1 -11575.232,E2 -11575.232} C_VEL
LIN {X 0,Y 414.899,Z 262.143,A -85,B 0,C 180,E1 -11577.284,E2 -11577.284} C_VEL
LIN {X 0,Y 409.985,Z 327.514,A -85,B 0,C 180,E1 -11579.111,E2 -11579.111} C_VEL
LIN {X 0,Y 408.043,Z 354.336,A -85,B 0,C 180,E1 -11579.894,E2 -11579.894} C_VEL
LIN {X 0,Y 405.957,Z 373.564,A -85,B 0,C 180,E1 -11580.649,E2 -11580.649} C_VEL
LIN {X 0,Y 404.331,Z 387.699,A -85,B 0,C 180,E1 -11581.374,E2 -11581.374} C_VEL
LIN {X 0,Y 402.158,Z 404.44,A -85,B 0,C 180,E1 -11582.412,E2 -11582.412} C_VEL
LIN {X 0,Y 399.951,Z 420.829,A -85,B 0,C 180,E1 -11583.66,E2 -11583.66} C_VEL
LIN {X 0,Y 397.857,Z 436.075,A -85,B 0,C 180,E1 -11585.055,E2 -11585.055} C_VEL
LIN {X 0,Y 395.74,Z 451.35,A -85,B 0,C 180,E1 -11586.725,E2 -11586.725} C_VEL
LIN {X 0,Y 393.854,Z 465.319,A -85,B 0,C 180,E1 -11588.542,E2 -11588.542} C_VEL
LIN {X 0,Y 392.375,Z 477.232,A -85,B 0,C 180,E1 -11590.376,E2 -11590.376} C_VEL
LIN {X 0,Y 391.125,Z 488.323,A -85,B 0,C 180,E1 -11592.376,E2 -11592.376} C_VEL
LIN {X 0,Y 390.101,Z 498.666,A -85,B 0,C 180,E1 -11594.589,E2 -11594.589} C_VEL
LIN {X 0,Y 389.474,Z 507.402,A -85,B 0,C 180,E1 -11596.842,E2 -11596.842} C_VEL
LIN {X 0,Y 389.027,Z 514.487,A -85,B 0,C 180,E1 -11599.065,E2 -11599.065} C_VEL
LIN {X 0,Y 388.85,Z 519.81,A -85,B 0,C 180,E1 -11601.162,E2 -11601.162} C_VEL
LIN {X 0,Y 388.905,Z 523.066,A -85,B 0,C 180,E1 -11602.732,E2 -11602.732} C_VEL
LIN {X 0,Y 388.88,Z 526.297,A -85,B 0,C 180,E1 -11604.815,E2 -11604.815} C_VEL
LIN {X 0,Y 388.963,Z 528.488,A -85,B 0,C 180,E1 -11606.892,E2 -11606.892} C_VEL
LIN {X 0,Y 388.994,Z 529.491,A -85,B 0,C 180,E1 -11608.964,E2 -11608.964} C_VEL
LIN {X 0,Y 388.995,Z 529.444,A -85,B 0,C 180,E1 -11611.035,E2 -11611.035} C_VEL
LIN {X 0,Y 388.977,Z 528.262,A -85,B 0,C 180,E1 -11613.106,E2 -11613.106} C_VEL
LIN {X 0,Y 388.892,Z 525.947,A -85,B 0,C 180,E1 -11615.184,E2 -11615.184} C_VEL
LIN {X 0,Y 388.911,Z 522.531,A -85,B 0,C 180,E1 -11617.266,E2 -11617.266} C_VEL
LIN {X 0,Y 388.899,Z 517.813,A -85,B 0,C 180,E1 -11619.36,E2 -11619.36} C_VEL
LIN {X 0,Y 389.124,Z 511.871,A -85,B 0,C 180,E1 -11621.459,E2 -11621.459} C_VEL
LIN {X 0,Y 389.521,Z 504.557,A -85,B 0,C 180,E1 -11623.565,E2 -11623.565} C_VEL
LIN {X 0,Y 390.187,Z 495.622,A -85,B 0,C 180,E1 -11625.674,E2 -11625.674} C_VEL
LIN {X 0,Y 391.017,Z 485.905,A -85,B 0,C 180,E1 -11627.6,E2 -11627.6} C_VEL
LIN {X 0,Y 392.049,Z 475.462,A -85,B 0,C 180,E1 -11629.367,E2 -11629.367} C_VEL
LIN {X 0,Y 393.324,Z 463.685,A -85,B 0,C 180,E1 -11631.074,E2 -11631.074} C_VEL
LIN {X 0,Y 394.854,Z 449.781,A -85,B 0,C 180,E1 -11632.775,E2 -11632.775} C_VEL
LIN {X 0,Y 396.321,Z 435.832,A -85,B 0,C 180,E1 -11634.209,E2 -11634.209} C_VEL
LIN {X 0,Y 397.959,Z 420.621,A -85,B 0,C 180,E1 -11635.511,E2 -11635.511} C_VEL
LIN {X 0,Y 399.35,Z 406.383,A -85,B 0,C 180,E1 -11636.523,E2 -11636.523} C_VEL
LIN {X 0,Y 400.811,Z 389.916,A -85,B 0,C 180,E1 -11637.475,E2 -11637.475} C_VEL
LIN {X 0,Y 402.122,Z 373.081,A -85,B 0,C 180,E1 -11638.227,E2 -11638.227} C_VEL
LIN {X 0,Y 403.209,Z 355.933,A -85,B 0,C 180,E1 -11638.783,E2 -11638.783} C_VEL
LIN {X 0,Y 409.342,Z 189.425,A -85,B 0,C 180,E1 -11642.522,E2 -11642.522} C_VEL
LIN {X 0,Y 404.19,Z 151.083,A -85,B 0,C 180,E1 -11643.886,E2 -11643.886} C_VEL
LIN {X 0,Y 403.02,Z 148.244,A -85,B 0,C 180,E1 -11644.077,E2 -11644.077} C_VEL
LIN {X 0,Y 397.711,Z 131.362,A -85,B 0,C 180,E1 -11646.483,E2 -11646.483} C_VEL
LIN {X 0,Y 390.717,Z 110.371,A -85,B 0,C 180,E1 -11649.663,E2 -11649.663} C_VEL
LIN {X 0,Y 390.092,Z 108.208,A -85,B 0,C 180,E1 -11650.031,E2 -11650.031} C_VEL
LIN {X 0,Y 390.109,Z 108.203,A -85,B 0,C 180,E1 -11653.202,E2 -11653.202} C_VEL
LIN {X 0,Y 390.054,Z 108.209,A -85,B 0,C 180,E1 -11656.789,E2 -11656.789} C_VEL
LIN {X 0,Y 390.052,Z 108.207,A -85,B 0,C 180,E1 -11659.56,E2 -11659.56} C_VEL
LIN {X 0,Y 390.041,Z 108.213,A -85,B 0,C 180,E1 -11662.448,E2 -11662.448} C_VEL
LIN {X 0,Y 390.079,Z 108.209,A -85,B 0,C 180,E1 -11666.047,E2 -11666.047} C_VEL
LIN {X 0,Y 390.039,Z 108.211,A -85,B 0,C 180,E1 -11669.701,E2 -11669.701} C_VEL
LIN {X 0,Y 390.109,Z 108.2,A -85,B 0,C 180,E1 -11673.232,E2 -11673.232} C_VEL
LIN {X 0,Y 390.102,Z 108.201,A -85,B 0,C 180,E1 -11676.75,E2 -11676.75} C_VEL
LIN {X 0,Y 390.099,Z 108.208,A -85,B 0,C 180,E1 -11679.983,E2 -11679.983} C_VEL
LIN {X 0,Y 390.137,Z 108.197,A -85,B 0,C 180,E1 -11683.248,E2 -11683.248} C_VEL
LIN {X 0,Y 390.19,Z 108.191,A -85,B 0,C 180,E1 -11686.561,E2 -11686.561} C_VEL
LIN {X 0,Y 390.173,Z 108.197,A -85,B 0,C 180,E1 -11689.623,E2 -11689.623} C_VEL
LIN {X 0,Y 390.314,Z 108.174,A -85,B 0,C 180,E1 -11692.759,E2 -11692.759} C_VEL
LIN {X 0,Y 390.223,Z 108.186,A -85,B 0,C 180,E1 -11694.834,E2 -11694.834} C_VEL
LIN {X 0,Y 390.416,Z 108.166,A -85,B 0,C 180,E1 -11697.937,E2 -11697.937} C_VEL
LIN {X 0,Y 390.546,Z 108.148,A -85,B 0,C 180,E1 -11700,E2 -11700} C_VEL
LIN {X 0,Y 390.311,Z 108.177,A -85,B 0,C 180,E1 -11703.097,E2 -11703.097} C_VEL
LIN {X 0,Y 390.305,Z 108.176,A -85,B 0,C 180,E1 -11706.642,E2 -11706.642} C_VEL
LIN {X 0,Y 390.2,Z 108.194,A -85,B 0,C 180,E1 -11709.329,E2 -11709.329} C_VEL
LIN {X 0,Y 390.166,Z 108.193,A -85,B 0,C 180,E1 -11712.483,E2 -11712.483} C_VEL
LIN {X 0,Y 390.135,Z 108.2,A -85,B 0,C 180,E1 -11715.677,E2 -11715.677} C_VEL
LIN {X 0,Y 390.101,Z 108.204,A -85,B 0,C 180,E1 -11718.922,E2 -11718.922} C_VEL
LIN {X 0,Y 390.036,Z 108.209,A -85,B 0,C 180,E1 -11722.234,E2 -11722.234} C_VEL
LIN {X 0,Y 390.115,Z 108.201,A -85,B 0,C 180,E1 -11725.744,E2 -11725.744} C_VEL
LIN {X 0,Y 390.055,Z 108.214,A -85,B 0,C 180,E1 -11729.11,E2 -11729.11} C_VEL
LIN {X 0,Y 390.039,Z 108.212,A -85,B 0,C 180,E1 -11732.722,E2 -11732.722} C_VEL
LIN {X 0,Y 390.053,Z 108.207,A -85,B 0,C 180,E1 -11735.826,E2 -11735.826} C_VEL
LIN {X 0,Y 390.068,Z 108.209,A -85,B 0,C 180,E1 -11739.219,E2 -11739.219} C_VEL
LIN {X 0,Y 390.041,Z 108.21,A -85,B 0,C 180,E1 -11742.375,E2 -11742.375} C_VEL
LIN {X 0,Y 390.045,Z 108.21,A -85,B 0,C 180,E1 -11745.356,E2 -11745.356} C_VEL
LIN {X 0,Y 390.066,Z 108.207,A -85,B 0,C 180,E1 -11748.192,E2 -11748.192} C_VEL
LIN {X 0,Y 390.089,Z 108.207,A -85,B 0,C 180,E1 -11750.909,E2 -11750.909} C_VEL
LIN {X 0,Y 390.082,Z 108.209,A -85,B 0,C 180,E1 -11754.794,E2 -11754.794} C_VEL
LIN {X 0,Y 390.022,Z 108.216,A -85,B 0,C 180,E1 -11758.496,E2 -11758.496} C_VEL
LIN {X 0,Y 390.115,Z 108.201,A -85,B 0,C 180,E1 -11762.071,E2 -11762.071} C_VEL
LIN {X 0,Y 390.078,Z 108.204,A -85,B 0,C 180,E1 -11765.52,E2 -11765.52} C_VEL
LIN {X 0,Y 390.071,Z 108.207,A -85,B 0,C 180,E1 -11768.879,E2 -11768.879} C_VEL
LIN {X 0,Y 390.13,Z 108.202,A -85,B 0,C 180,E1 -11772.168,E2 -11772.168} C_VEL
LIN {X 0,Y 390.143,Z 108.196,A -85,B 0,C 180,E1 -11775.393,E2 -11775.393} C_VEL
LIN {X 0,Y 390.148,Z 108.198,A -85,B 0,C 180,E1 -11778.572,E2 -11778.572} C_VEL
LIN {X 0,Y 390.344,Z 108.175,A -85,B 0,C 180,E1 -11781.994,E2 -11781.994} C_VEL
LIN {X 0,Y 390.227,Z 108.186,A -85,B 0,C 180,E1 -11784.834,E2 -11784.834} C_VEL
LIN {X 0,Y 390.419,Z 108.166,A -85,B 0,C 180,E1 -11787.937,E2 -11787.937} C_VEL
LIN {X 0,Y 390.549,Z 108.152,A -85,B 0,C 180,E1 -11790.001,E2 -11790.001} C_VEL
LIN {X 0,Y 390.311,Z 108.175,A -85,B 0,C 180,E1 -11793.097,E2 -11793.097} C_VEL
LIN {X 0,Y 390.331,Z 108.176,A -85,B 0,C 180,E1 -11796.203,E2 -11796.203} C_VEL
LIN {X 0,Y 390.316,Z 108.177,A -85,B 0,C 180,E1 -11798.283,E2 -11798.283} C_VEL
LIN {X 0,Y 390.172,Z 108.193,A -85,B 0,C 180,E1 -11802.484,E2 -11802.484} C_VEL
LIN {X 0,Y 390.141,Z 108.202,A -85,B 0,C 180,E1 -11805.677,E2 -11805.677} C_VEL
LIN {X 0,Y 390.108,Z 108.2,A -85,B 0,C 180,E1 -11808.923,E2 -11808.923} C_VEL
LIN {X 0,Y 390.041,Z 108.21,A -85,B 0,C 180,E1 -11812.235,E2 -11812.235} C_VEL
LIN {X 0,Y 390.121,Z 108.204,A -85,B 0,C 180,E1 -11815.744,E2 -11815.744} C_VEL
LIN {X 0,Y 390.061,Z 108.208,A -85,B 0,C 180,E1 -11819.11,E2 -11819.11} C_VEL
LIN {X 0,Y 390.014,Z 108.212,A -85,B 0,C 180,E1 -11820.809,E2 -11820.809} C_VEL
LIN {X 0,Y 389.341,Z 108.301,A -85,B 0,C 180,E1 -11821.671,E2 -11821.671} C_VEL
LIN {X 0,Y 386.494,Z 108.653,A -85,B 0,C 180,E1 -11823.072,E2 -11823.072} C_VEL
LIN {X 0,Y 384.096,Z 108.95,A -85,B 0,C 180,E1 -11824.205,E2 -11824.205} C_VEL
LIN {X 0,Y 383.077,Z 109.079,A -85,B 0,C 180,E1 -11825.081,E2 -11825.081} C_VEL
LIN {X 0,Y 383,Z 109.084,A -85,B 0,C 180,E1 -11825.378,E2 -11825.378} C_VEL
LIN {X 0,Y 383.006,Z 109.085,A -85,B 0,C 180,E1 -11828.601,E2 -11828.601} C_VEL
LIN {X 0,Y 382.988,Z 109.094,A -85,B 0,C 180,E1 -11831.348,E2 -11831.348} C_VEL
LIN {X 0,Y 383.001,Z 109.085,A -85,B 0,C 180,E1 -11834.304,E2 -11834.304} C_VEL
LIN {X 0,Y 383.013,Z 109.091,A -85,B 0,C 180,E1 -11837.241,E2 -11837.241} C_VEL
LIN {X 0,Y 383.017,Z 109.084,A -85,B 0,C 180,E1 -11840.414,E2 -11840.414} C_VEL
LIN {X 0,Y 383.028,Z 109.086,A -85,B 0,C 180,E1 -11844.045,E2 -11844.045} C_VEL
LIN {X 0,Y 383.063,Z 109.082,A -85,B 0,C 180,E1 -11845.044,E2 -11845.044} C_VEL
LIN {X 0,Y 384.097,Z 111.968,A -85,B 0,C 180,E1 -11845.224,E2 -11845.224} C_VEL
LIN {X 0,Y 402.086,Z 147.62,A -85,B 0,C 180,E1 -11847.589,E2 -11847.589} C_VEL
LIN {X 0,Y 402.558,Z 148.586,A -85,B 0,C 180,E1 -11847.649,E2 -11847.649} C_VEL
LIN {X 0,Y 397.213,Z 289.139,A -85,B 0,C 180,E1 -11850.849,E2 -11850.849} C_VEL
LIN {X 0,Y 396.463,Z 307.398,A -85,B 0,C 180,E1 -11851.368,E2 -11851.368} C_VEL
LIN {X 0,Y 395.53,Z 324.118,A -85,B 0,C 180,E1 -11852.054,E2 -11852.054} C_VEL
LIN {X 0,Y 394.359,Z 340.756,A -85,B 0,C 180,E1 -11852.945,E2 -11852.945} C_VEL
LIN {X 0,Y 393.064,Z 356.723,A -85,B 0,C 180,E1 -11854.02,E2 -11854.02} C_VEL
LIN {X 0,Y 391.703,Z 371.234,A -85,B 0,C 180,E1 -11855.203,E2 -11855.203} C_VEL
LIN {X 0,Y 390.276,Z 384.874,A -85,B 0,C 180,E1 -11856.52,E2 -11856.52} C_VEL
LIN {X 0,Y 388.776,Z 398.72,A -85,B 0,C 180,E1 -11858.109,E2 -11858.109} C_VEL
LIN {X 0,Y 387.298,Z 411.379,A -85,B 0,C 180,E1 -11859.832,E2 -11859.832} C_VEL
LIN {X 0,Y 386.198,Z 421.933,A -85,B 0,C 180,E1 -11861.523,E2 -11861.523} C_VEL
LIN {X 0,Y 384.956,Z 432.826,A -85,B 0,C 180,E1 -11863.562,E2 -11863.562} C_VEL
LIN {X 0,Y 384.01,Z 442.359,A -85,B 0,C 180,E1 -11865.696,E2 -11865.696} C_VEL
LIN {X 0,Y 383.237,Z 450.292,A -85,B 0,C 180,E1 -11867.825,E2 -11867.825} C_VEL
LIN {X 0,Y 382.684,Z 456.769,A -85,B 0,C 180,E1 -11869.952,E2 -11869.952} C_VEL
LIN {X 0,Y 382.378,Z 461.956,A -85,B 0,C 180,E1 -11872.077,E2 -11872.077} C_VEL
LIN {X 0,Y 382.183,Z 465.101,A -85,B 0,C 180,E1 -11873.665,E2 -11873.665} C_VEL
LIN {X 0,Y 382.04,Z 468.3,A -85,B 0,C 180,E1 -11875.78,E2 -11875.78} C_VEL
LIN {X 0,Y 381.974,Z 470.47,A -85,B 0,C 180,E1 -11877.891,E2 -11877.891} C_VEL
LIN {X 0,Y 381.923,Z 471.542,A -85,B 0,C 180,E1 -11880,E2 -11880} C_VEL
LIN {X 0,Y 382.098,Z 471.657,A -85,B 0,C 180,E1 -11882.108,E2 -11882.108} C_VEL
LIN {X 0,Y 382.259,Z 470.672,A -85,B 0,C 180,E1 -11884.217,E2 -11884.217} C_VEL
LIN {X 0,Y 382.35,Z 468.732,A -85,B 0,C 180,E1 -11886.332,E2 -11886.332} C_VEL
LIN {X 0,Y 382.927,Z 465.687,A -85,B 0,C 180,E1 -11888.443,E2 -11888.443} C_VEL
LIN {X 0,Y 383.56,Z 461.531,A -85,B 0,C 180,E1 -11890.558,E2 -11890.558} C_VEL
LIN {X 0,Y 384.312,Z 456.273,A -85,B 0,C 180,E1 -11892.676,E2 -11892.676} C_VEL
LIN {X 0,Y 385.395,Z 449.448,A -85,B 0,C 180,E1 -11894.871,E2 -11894.871} C_VEL
LIN {X 0,Y 386.647,Z 441.714,A -85,B 0,C 180,E1 -11896.907,E2 -11896.907} C_VEL
LIN {X 0,Y 388.299,Z 432.12,A -85,B 0,C 180,E1 -11899.013,E2 -11899.013} C_VEL
LIN {X 0,Y 390.03,Z 422.199,A -85,B 0,C 180,E1 -11900.847,E2 -11900.847} C_VEL
LIN {X 0,Y 391.985,Z 410.567,A -85,B 0,C 180,E1 -11902.673,E2 -11902.673} C_VEL
LIN {X 0,Y 393.764,Z 399.9,A -85,B 0,C 180,E1 -11904.097,E2 -11904.097} C_VEL
LIN {X 0,Y 395.916,Z 386.387,A -85,B 0,C 180,E1 -11905.638,E2 -11905.638} C_VEL
LIN {X 0,Y 397.812,Z 373.205,A -85,B 0,C 180,E1 -11906.917,E2 -11906.917} C_VEL
LIN {X 0,Y 399.742,Z 359.124,A -85,B 0,C 180,E1 -11908.066,E2 -11908.066} C_VEL
LIN {X 0,Y 401.683,Z 342.86,A -85,B 0,C 180,E1 -11909.161,E2 -11909.161} C_VEL
LIN {X 0,Y 403.316,Z 326.199,A -85,B 0,C 180,E1 -11910.065,E2 -11910.065} C_VEL
LIN {X 0,Y 404.763,Z 308.971,A -85,B 0,C 180,E1 -11910.775,E2 -11910.775} C_VEL
LIN {X 0,Y 407.332,Z 276.358,A -85,B 0,C 180,E1 -11911.751,E2 -11911.751} C_VEL
LIN {X 0,Y 413.619,Z 211.778,A -85,B 0,C 180,E1 -11913.702,E2 -11913.702} C_VEL
LIN {X 0,Y 419.808,Z 159.872,A -85,B 0,C 180,E1 -11915.31,E2 -11915.31} C_VEL
LIN {X 0,Y 417.139,Z 154.497,A -85,B 0,C 180,E1 -11916.288,E2 -11916.288} C_VEL
LIN {X 0,Y 413.973,Z 149.766,A -85,B 0,C 180,E1 -11917.521,E2 -11917.521} C_VEL
LIN {X 0,Y 410.797,Z 145.349,A -85,B 0,C 180,E1 -11919.056,E2 -11919.056} C_VEL
LIN {X 0,Y 407.692,Z 142.087,A -85,B 0,C 180,E1 -11921.137,E2 -11921.137} C_VEL
LIN {X 0,Y 406.531,Z 141.138,A -85,B 0,C 180,E1 -11922.393,E2 -11922.393} C_VEL
LIN {X 0,Y 405.782,Z 141.275,A -85,B 0,C 180,E1 -11923.993,E2 -11923.993} C_VEL
LIN {X 0,Y 405.961,Z 143.028,A -85,B 0,C 180,E1 -11925.871,E2 -11925.871} C_VEL
LIN {X 0,Y 406.979,Z 145.342,A -85,B 0,C 180,E1 -11927.349,E2 -11927.349} C_VEL
LIN {X 0,Y 408.278,Z 148.22,A -85,B 0,C 180,E1 -11928.541,E2 -11928.541} C_VEL
LIN {X 0,Y 411.249,Z 154.646,A -85,B 0,C 180,E1 -11930.435,E2 -11930.435} C_VEL
LIN {X 0,Y 414.663,Z 162.642,A -85,B 0,C 180,E1 -11932.077,E2 -11932.077} C_VEL
LIN {X 0,Y 416.901,Z 168.707,A -85,B 0,C 180,E1 -11933.021,E2 -11933.021} C_VEL
LIN {X 0,Y 417.121,Z 181.294,A -85,B 0,C 180,E1 -11933.809,E2 -11933.809} C_VEL
LIN {X 0,Y 417.137,Z 194.202,A -85,B 0,C 180,E1 -11934.514,E2 -11934.514} C_VEL
LIN {X 0,Y 409.87,Z 263.787,A -85,B 0,C 180,E1 -11936.611,E2 -11936.611} C_VEL
LIN {X 0,Y 404.496,Z 329.337,A -85,B 0,C 180,E1 -11938.511,E2 -11938.511} C_VEL
LIN {X 0,Y 402.55,Z 353.373,A -85,B 0,C 180,E1 -11939.238,E2 -11939.238} C_VEL
LIN {X 0,Y 400.581,Z 370.668,A -85,B 0,C 180,E1 -11939.926,E2 -11939.926} C_VEL
LIN {X 0,Y 398.625,Z 386.13,A -85,B 0,C 180,E1 -11940.708,E2 -11940.708} C_VEL
LIN {X 0,Y 396.165,Z 403.699,A -85,B 0,C 180,E1 -11941.814,E2 -11941.814} C_VEL
LIN {X 0,Y 393.791,Z 420.442,A -85,B 0,C 180,E1 -11943.121,E2 -11943.121} C_VEL
LIN {X 0,Y 391.606,Z 435.127,A -85,B 0,C 180,E1 -11944.486,E2 -11944.486} C_VEL
LIN {X 0,Y 389.348,Z 450.367,A -85,B 0,C 180,E1 -11946.178,E2 -11946.178} C_VEL
LIN {X 0,Y 387.353,Z 463.955,A -85,B 0,C 180,E1 -11947.969,E2 -11947.969} C_VEL
LIN {X 0,Y 385.578,Z 477.068,A -85,B 0,C 180,E1 -11950.015,E2 -11950.015} C_VEL
LIN {X 0,Y 384.279,Z 487.768,A -85,B 0,C 180,E1 -11951.992,E2 -11951.992} C_VEL
LIN {X 0,Y 383.265,Z 497.208,A -85,B 0,C 180,E1 -11954.034,E2 -11954.034} C_VEL
LIN {X 0,Y 382.543,Z 505.607,A -85,B 0,C 180,E1 -11956.182,E2 -11956.182} C_VEL
LIN {X 0,Y 382.031,Z 512.51,A -85,B 0,C 180,E1 -11958.324,E2 -11958.324} C_VEL
LIN {X 0,Y 381.788,Z 518.126,A -85,B 0,C 180,E1 -11960.463,E2 -11960.463} C_VEL
LIN {X 0,Y 381.815,Z 522.594,A -85,B 0,C 180,E1 -11962.596,E2 -11962.596} C_VEL
LIN {X 0,Y 381.8,Z 525.792,A -85,B 0,C 180,E1 -11964.718,E2 -11964.718} C_VEL
LIN {X 0,Y 381.878,Z 527.942,A -85,B 0,C 180,E1 -11966.834,E2 -11966.834} C_VEL
LIN {X 0,Y 381.927,Z 528.933,A -85,B 0,C 180,E1 -11968.945,E2 -11968.945} C_VEL
LIN {X 0,Y 381.945,Z 528.836,A -85,B 0,C 180,E1 -11971.054,E2 -11971.054} C_VEL
LIN {X 0,Y 381.911,Z 527.626,A -85,B 0,C 180,E1 -11973.164,E2 -11973.164} C_VEL
LIN {X 0,Y 381.835,Z 525.247,A -85,B 0,C 180,E1 -11975.28,E2 -11975.28} C_VEL
LIN {X 0,Y 381.829,Z 521.776,A -85,B 0,C 180,E1 -11977.402,E2 -11977.402} C_VEL
LIN {X 0,Y 381.834,Z 516.991,A -85,B 0,C 180,E1 -11979.534,E2 -11979.534} C_VEL
LIN {X 0,Y 382.065,Z 510.951,A -85,B 0,C 180,E1 -11981.673,E2 -11981.673} C_VEL
LIN {X 0,Y 382.495,Z 503.528,A -85,B 0,C 180,E1 -11983.819,E2 -11983.819} C_VEL
LIN {X 0,Y 383.218,Z 494.517,A -85,B 0,C 180,E1 -11985.967,E2 -11985.967} C_VEL
LIN {X 0,Y 384.174,Z 483.645,A -85,B 0,C 180,E1 -11988.118,E2 -11988.118} C_VEL
LIN {X 0,Y 385.336,Z 472.338,A -85,B 0,C 180,E1 -11989.996,E2 -11989.996} C_VEL
LIN {X 0,Y 386.789,Z 459.687,A -85,B 0,C 180,E1 -11991.778,E2 -11991.778} C_VEL
LIN {X 0,Y 388.241,Z 446.752,A -85,B 0,C 180,E1 -11993.327,E2 -11993.327} C_VEL
LIN {X 0,Y 389.839,Z 432.386,A -85,B 0,C 180,E1 -11994.78,E2 -11994.78} C_VEL
LIN {X 0,Y 391.475,Z 417.233,A -85,B 0,C 180,E1 -11996.058,E2 -11996.058} C_VEL
LIN {X 0,Y 393.16,Z 400.741,A -85,B 0,C 180,E1 -11997.189,E2 -11997.189} C_VEL
LIN {X 0,Y 394.586,Z 384.242,A -85,B 0,C 180,E1 -11998.091,E2 -11998.091} C_VEL
LIN {X 0,Y 395.844,Z 367.351,A -85,B 0,C 180,E1 -11998.788,E2 -11998.788} C_VEL
LIN {X 0,Y 396.825,Z 350.19,A -85,B 0,C 180,E1 -11999.291,E2 -11999.291} C_VEL
LIN {X 0,Y 402.967,Z 190.346,A -85,B 0,C 180,E1 -12002.95,E2 -12002.95} C_VEL
LIN {X 0,Y 398.164,Z 153.756,A -85,B 0,C 180,E1 -12004.282,E2 -12004.282} C_VEL
LIN {X 0,Y 395.656,Z 148.015,A -85,B 0,C 180,E1 -12004.639,E2 -12004.639} C_VEL
LIN {X 0,Y 390.282,Z 131.268,A -85,B 0,C 180,E1 -12007.083,E2 -12007.083} C_VEL
LIN {X 0,Y 383.725,Z 111.32,A -85,B 0,C 180,E1 -12010.163,E2 -12010.163} C_VEL
LIN {X 0,Y 383.04,Z 109.087,A -85,B 0,C 180,E1 -12010.525,E2 -12010.525} C_VEL
LIN {X 0,Y 383.061,Z 109.084,A -85,B 0,C 180,E1 -12012.788,E2 -12012.788} C_VEL
LIN {X 0,Y 383.003,Z 109.09,A -85,B 0,C 180,E1 -12015.79,E2 -12015.79} C_VEL
LIN {X 0,Y 382.984,Z 109.09,A -85,B 0,C 180,E1 -12018.795,E2 -12018.795} C_VEL
LIN {X 0,Y 382.997,Z 109.09,A -85,B 0,C 180,E1 -12022.095,E2 -12022.095} C_VEL
LIN {X 0,Y 383.013,Z 109.084,A -85,B 0,C 180,E1 -12025.332,E2 -12025.332} C_VEL
LIN {X 0,Y 383.032,Z 109.085,A -85,B 0,C 180,E1 -12027.853,E2 -12027.853} C_VEL
LIN {X 0,Y 383.059,Z 109.081,A -85,B 0,C 180,E1 -12031.72,E2 -12031.72} C_VEL
LIN {X 0,Y 383.047,Z 109.08,A -85,B 0,C 180,E1 -12035.04,E2 -12035.04} C_VEL
LIN {X 0,Y 382.988,Z 109.089,A -85,B 0,C 180,E1 -12038.469,E2 -12038.469} C_VEL
LIN {X 0,Y 383.085,Z 109.08,A -85,B 0,C 180,E1 -12041.828,E2 -12041.828} C_VEL
LIN {X 0,Y 383.11,Z 109.072,A -85,B 0,C 180,E1 -12045.118,E2 -12045.118} C_VEL
LIN {X 0,Y 383.102,Z 109.074,A -85,B 0,C 180,E1 -12048.358,E2 -12048.358} C_VEL
LIN {X 0,Y 383.299,Z 109.053,A -85,B 0,C 180,E1 -12051.933,E2 -12051.933} C_VEL
LIN {X 0,Y 383.195,Z 109.061,A -85,B 0,C 180,E1 -12054.739,E2 -12054.739} C_VEL
LIN {X 0,Y 383.383,Z 109.042,A -85,B 0,C 180,E1 -12057.899,E2 -12057.899} C_VEL
LIN {X 0,Y 383.515,Z 109.024,A -85,B 0,C 180,E1 -12060,E2 -12060} C_VEL
LIN {X 0,Y 383.247,Z 109.057,A -85,B 0,C 180,E1 -12063.154,E2 -12063.154} C_VEL
LIN {X 0,Y 383.265,Z 109.053,A -85,B 0,C 180,E1 -12066.637,E2 -12066.637} C_VEL
LIN {X 0,Y 383.255,Z 109.054,A -85,B 0,C 180,E1 -12068.436,E2 -12068.436} C_VEL
LIN {X 0,Y 383.093,Z 109.078,A -85,B 0,C 180,E1 -12071.642,E2 -12071.642} C_VEL
LIN {X 0,Y 383.106,Z 109.074,A -85,B 0,C 180,E1 -12074.882,E2 -12074.882} C_VEL
LIN {X 0,Y 383.059,Z 109.078,A -85,B 0,C 180,E1 -12078.174,E2 -12078.174} C_VEL
LIN {X 0,Y 382.989,Z 109.091,A -85,B 0,C 180,E1 -12081.531,E2 -12081.531} C_VEL
LIN {X 0,Y 383.048,Z 109.084,A -85,B 0,C 180,E1 -12084.961,E2 -12084.961} C_VEL
LIN {X 0,Y 383.025,Z 109.083,A -85,B 0,C 180,E1 -12088.271,E2 -12088.271} C_VEL
LIN {X 0,Y 383.005,Z 109.085,A -85,B 0,C 180,E1 -12092.15,E2 -12092.15} C_VEL
LIN {X 0,Y 383.014,Z 109.087,A -85,B 0,C 180,E1 -12094.668,E2 -12094.668} C_VEL
LIN {X 0,Y 382.998,Z 109.086,A -85,B 0,C 180,E1 -12097.905,E2 -12097.905} C_VEL
LIN {X 0,Y 382.981,Z 109.09,A -85,B 0,C 180,E1 -12101.348,E2 -12101.348} C_VEL
LIN {X 0,Y 382.996,Z 109.087,A -85,B 0,C 180,E1 -12104.305,E2 -12104.305} C_VEL
LIN {X 0,Y 383.036,Z 109.083,A -85,B 0,C 180,E1 -12107.245,E2 -12107.245} C_VEL
LIN {X 0,Y 383.017,Z 109.087,A -85,B 0,C 180,E1 -12110.413,E2 -12110.413} C_VEL
LIN {X 0,Y 383.022,Z 109.084,A -85,B 0,C 180,E1 -12114.045,E2 -12114.045} C_VEL
LIN {X 0,Y 382.984,Z 109.088,A -85,B 0,C 180,E1 -12117.579,E2 -12117.579} C_VEL
LIN {X 0,Y 382.99,Z 109.09,A -85,B 0,C 180,E1 -12120.301,E2 -12120.301} C_VEL
LIN {X 0,Y 383.079,Z 109.078,A -85,B 0,C 180,E1 -12124.021,E2 -12124.021} C_VEL
LIN {X 0,Y 383.012,Z 109.084,A -85,B 0,C 180,E1 -12127.336,E2 -12127.336} C_VEL
LIN {X 0,Y 383.071,Z 109.08,A -85,B 0,C 180,E1 -12130.718,E2 -12130.718} C_VEL
LIN {X 0,Y 383.08,Z 109.079,A -85,B 0,C 180,E1 -12134.027,E2 -12134.027} C_VEL
LIN {X 0,Y 383.136,Z 109.069,A -85,B 0,C 180,E1 -12137.285,E2 -12137.285} C_VEL
LIN {X 0,Y 383.155,Z 109.07,A -85,B 0,C 180,E1 -12140.499,E2 -12140.499} C_VEL
LIN {X 0,Y 383.274,Z 109.054,A -85,B 0,C 180,E1 -12142.626,E2 -12142.626} C_VEL
LIN {X 0,Y 383.199,Z 109.062,A -85,B 0,C 180,E1 -12144.739,E2 -12144.739} C_VEL
LIN {X 0,Y 383.386,Z 109.042,A -85,B 0,C 180,E1 -12147.9,E2 -12147.9} C_VEL
LIN {X 0,Y 383.518,Z 109.027,A -85,B 0,C 180,E1 -12150.001,E2 -12150.001} C_VEL
LIN {X 0,Y 383.247,Z 109.055,A -85,B 0,C 180,E1 -12153.154,E2 -12153.154} C_VEL
LIN {X 0,Y 383.288,Z 109.052,A -85,B 0,C 180,E1 -12156.317,E2 -12156.317} C_VEL
LIN {X 0,Y 383.261,Z 109.055,A -85,B 0,C 180,E1 -12158.436,E2 -12158.436} C_VEL
LIN {X 0,Y 383.099,Z 109.078,A -85,B 0,C 180,E1 -12161.643,E2 -12161.643} C_VEL
LIN {X 0,Y 383.112,Z 109.072,A -85,B 0,C 180,E1 -12164.882,E2 -12164.882} C_VEL
LIN {X 0,Y 383.065,Z 109.08,A -85,B 0,C 180,E1 -12168.174,E2 -12168.174} C_VEL
LIN {X 0,Y 382.995,Z 109.091,A -85,B 0,C 180,E1 -12171.532,E2 -12171.532} C_VEL
LIN {X 0,Y 383.054,Z 109.08,A -85,B 0,C 180,E1 -12174.961,E2 -12174.961} C_VEL
LIN {X 0,Y 383.032,Z 109.082,A -85,B 0,C 180,E1 -12178.271,E2 -12178.271} C_VEL
LIN {X 0,Y 383.012,Z 109.085,A -85,B 0,C 180,E1 -12182.15,E2 -12182.15} C_VEL
LIN {X 0,Y 383,Z 109.084,A -85,B 0,C 180,E1 -12185.378,E2 -12185.378} C_VEL
LIN {X 0,Y 382.363,Z 109.166,A -85,B 0,C 180,E1 -12186.255,E2 -12186.255} C_VEL
LIN {X 0,Y 379.567,Z 109.517,A -85,B 0,C 180,E1 -12187.684,E2 -12187.684} C_VEL
LIN {X 0,Y 377.163,Z 109.817,A -85,B 0,C 180,E1 -12188.838,E2 -12188.838} C_VEL
LIN {X 0,Y 376.092,Z 109.95,A -85,B 0,C 180,E1 -12189.73,E2 -12189.73} C_VEL
LIN {X 0,Y 375.985,Z 109.96,A -85,B 0,C 180,E1 -12190.032,E2 -12190.032} C_VEL
LIN {X 0,Y 375.934,Z 109.968,A -85,B 0,C 180,E1 -12193.766,E2 -12193.766} C_VEL
LIN {X 0,Y 375.937,Z 109.968,A -85,B 0,C 180,E1 -12196.811,E2 -12196.811} C_VEL
LIN {X 0,Y 375.965,Z 109.963,A -85,B 0,C 180,E1 -12200.538,E2 -12200.538} C_VEL
LIN {X 0,Y 376.025,Z 110.082,A -85,B 0,C 180,E1 -12204.491,E2 -12204.491} C_VEL
LIN {X 0,Y 377.12,Z 112.977,A -85,B 0,C 180,E1 -12204.669,E2 -12204.669} C_VEL
LIN {X 0,Y 393.2,Z 144.818,A -85,B 0,C 180,E1 -12206.855,E2 -12206.855} C_VEL
LIN {X 0,Y 396.164,Z 150.722,A -85,B 0,C 180,E1 -12207.237,E2 -12207.237} C_VEL
LIN {X 0,Y 390.252,Z 299.198,A -85,B 0,C 180,E1 -12210.722,E2 -12210.722} C_VEL
LIN {X 0,Y 389.405,Z 316.864,A -85,B 0,C 180,E1 -12211.354,E2 -12211.354} C_VEL
LIN {X 0,Y 388.322,Z 333.154,A -85,B 0,C 180,E1 -12212.141,E2 -12212.141} C_VEL
LIN {X 0,Y 387.193,Z 347.519,A -85,B 0,C 180,E1 -12213.014,E2 -12213.014} C_VEL
LIN {X 0,Y 385.753,Z 363.712,A -85,B 0,C 180,E1 -12214.216,E2 -12214.216} C_VEL
LIN {X 0,Y 384.177,Z 378.586,A -85,B 0,C 180,E1 -12215.55,E2 -12215.55} C_VEL
LIN {X 0,Y 382.56,Z 393.096,A -85,B 0,C 180,E1 -12217.112,E2 -12217.112} C_VEL
LIN {X 0,Y 381.206,Z 405.159,A -85,B 0,C 180,E1 -12218.647,E2 -12218.647} C_VEL
LIN {X 0,Y 379.869,Z 416.094,A -85,B 0,C 180,E1 -12220.266,E2 -12220.266} C_VEL
LIN {X 0,Y 378.716,Z 427.095,A -85,B 0,C 180,E1 -12222.17,E2 -12222.17} C_VEL
LIN {X 0,Y 377.606,Z 436.504,A -85,B 0,C 180,E1 -12224.066,E2 -12224.066} C_VEL
LIN {X 0,Y 376.711,Z 445.517,A -85,B 0,C 180,E1 -12226.239,E2 -12226.239} C_VEL
LIN {X 0,Y 376.033,Z 452.097,A -85,B 0,C 180,E1 -12228.136,E2 -12228.136} C_VEL
LIN {X 0,Y 375.573,Z 458.389,A -85,B 0,C 180,E1 -12230.304,E2 -12230.304} C_VEL
LIN {X 0,Y 375.284,Z 463.385,A -85,B 0,C 180,E1 -12232.467,E2 -12232.467} C_VEL
LIN {X 0,Y 374.979,Z 467.206,A -85,B 0,C 180,E1 -12234.623,E2 -12234.623} C_VEL
LIN {X 0,Y 374.985,Z 469.986,A -85,B 0,C 180,E1 -12236.777,E2 -12236.777} C_VEL
LIN {X 0,Y 374.837,Z 471.643,A -85,B 0,C 180,E1 -12238.926,E2 -12238.926} C_VEL
LIN {X 0,Y 374.918,Z 472.321,A -85,B 0,C 180,E1 -12241.074,E2 -12241.074} C_VEL
LIN {X 0,Y 375.198,Z 471.936,A -85,B 0,C 180,E1 -12243.221,E2 -12243.221} C_VEL
LIN {X 0,Y 375.346,Z 470.543,A -85,B 0,C 180,E1 -12245.372,E2 -12245.372} C_VEL
LIN {X 0,Y 375.68,Z 468.152,A -85,B 0,C 180,E1 -12247.524,E2 -12247.524} C_VEL
LIN {X 0,Y 376.414,Z 463.594,A -85,B 0,C 180,E1 -12250.217,E2 -12250.217} C_VEL
LIN {X 0,Y 377.223,Z 458.637,A -85,B 0,C 180,E1 -12252.372,E2 -12252.372} C_VEL
LIN {X 0,Y 378.121,Z 452.976,A -85,B 0,C 180,E1 -12254.384,E2 -12254.384} C_VEL
LIN {X 0,Y 379.572,Z 445.029,A -85,B 0,C 180,E1 -12256.678,E2 -12256.678} C_VEL
LIN {X 0,Y 381.212,Z 435.989,A -85,B 0,C 180,E1 -12258.822,E2 -12258.822} C_VEL
LIN {X 0,Y 382.906,Z 427.07,A -85,B 0,C 180,E1 -12260.596,E2 -12260.596} C_VEL
LIN {X 0,Y 385.025,Z 415.627,A -85,B 0,C 180,E1 -12262.539,E2 -12262.539} C_VEL
LIN {X 0,Y 387.294,Z 402.726,A -85,B 0,C 180,E1 -12264.383,E2 -12264.383} C_VEL
LIN {X 0,Y 389.803,Z 388.472,A -85,B 0,C 180,E1 -12266.07,E2 -12266.07} C_VEL
LIN {X 0,Y 391.822,Z 375.656,A -85,B 0,C 180,E1 -12267.363,E2 -12267.363} C_VEL
LIN {X 0,Y 393.793,Z 362.172,A -85,B 0,C 180,E1 -12268.516,E2 -12268.516} C_VEL
LIN {X 0,Y 395.997,Z 345.681,A -85,B 0,C 180,E1 -12269.676,E2 -12269.676} C_VEL
LIN {X 0,Y 397.902,Z 328.295,A -85,B 0,C 180,E1 -12270.664,E2 -12270.664} C_VEL
LIN {X 0,Y 399.553,Z 310.258,A -85,B 0,C 180,E1 -12271.442,E2 -12271.442} C_VEL
LIN {X 0,Y 402.656,Z 274.973,A -85,B 0,C 180,E1 -12272.534,E2 -12272.534} C_VEL
LIN {X 0,Y 409.522,Z 211.141,A -85,B 0,C 180,E1 -12274.528,E2 -12274.528} C_VEL
LIN {X 0,Y 415.692,Z 163.43,A -85,B 0,C 180,E1 -12276.048,E2 -12276.048} C_VEL
LIN {X 0,Y 413.48,Z 159.248,A -85,B 0,C 180,E1 -12276.928,E2 -12276.928} C_VEL
LIN {X 0,Y 411.04,Z 155.512,A -85,B 0,C 180,E1 -12277.99,E2 -12277.99} C_VEL
LIN {X 0,Y 408.574,Z 151.965,A -85,B 0,C 180,E1 -12279.28,E2 -12279.28} C_VEL
LIN {X 0,Y 405.854,Z 148.9,A -85,B 0,C 180,E1 -12281.213,E2 -12281.213} C_VEL
LIN {X 0,Y 404.624,Z 147.978,A -85,B 0,C 180,E1 -12282.64,E2 -12282.64} C_VEL
LIN {X 0,Y 404.014,Z 148.247,A -85,B 0,C 180,E1 -12284.092,E2 -12284.092} C_VEL
LIN {X 0,Y 404.224,Z 150.077,A -85,B 0,C 180,E1 -12285.936,E2 -12285.936} C_VEL
LIN {X 0,Y 405.375,Z 152.769,A -85,B 0,C 180,E1 -12287.545,E2 -12287.545} C_VEL
LIN {X 0,Y 407.239,Z 157.524,A -85,B 0,C 180,E1 -12289.174,E2 -12289.174} C_VEL
LIN {X 0,Y 409.286,Z 162.351,A -85,B 0,C 180,E1 -12290.444,E2 -12290.444} C_VEL
LIN {X 0,Y 411.739,Z 168.675,A -85,B 0,C 180,E1 -12291.712,E2 -12291.712} C_VEL
LIN {X 0,Y 413.178,Z 172.709,A -85,B 0,C 180,E1 -12292.376,E2 -12292.376} C_VEL
LIN {X 0,Y 413.078,Z 190.508,A -85,B 0,C 180,E1 -12293.477,E2 -12293.477} C_VEL
LIN {X 0,Y 412.847,Z 196.214,A -85,B 0,C 180,E1 -12293.764,E2 -12293.764} C_VEL
LIN {X 0,Y 405.023,Z 265.048,A -85,B 0,C 180,E1 -12295.896,E2 -12295.896} C_VEL
LIN {X 0,Y 398.962,Z 332.987,A -85,B 0,C 180,E1 -12297.926,E2 -12297.926} C_VEL
LIN {X 0,Y 396.992,Z 354.551,A -85,B 0,C 180,E1 -12298.62,E2 -12298.62} C_VEL
LIN {X 0,Y 394.604,Z 373.504,A -85,B 0,C 180,E1 -12299.422,E2 -12299.422} C_VEL
LIN {X 0,Y 392.731,Z 386.967,A -85,B 0,C 180,E1 -12300.151,E2 -12300.151} C_VEL
LIN {X 0,Y 390.027,Z 404.915,A -85,B 0,C 180,E1 -12301.329,E2 -12301.329} C_VEL
LIN {X 0,Y 387.536,Z 421.031,A -85,B 0,C 180,E1 -12302.634,E2 -12302.634} C_VEL
LIN {X 0,Y 385.204,Z 435.557,A -85,B 0,C 180,E1 -12304.031,E2 -12304.031} C_VEL
LIN {X 0,Y 382.811,Z 450.558,A -85,B 0,C 180,E1 -12305.745,E2 -12305.745} C_VEL
LIN {X 0,Y 380.643,Z 464.503,A -85,B 0,C 180,E1 -12307.638,E2 -12307.638} C_VEL
LIN {X 0,Y 378.799,Z 476.986,A -85,B 0,C 180,E1 -12309.642,E2 -12309.642} C_VEL
LIN {X 0,Y 377.329,Z 488.243,A -85,B 0,C 180,E1 -12311.787,E2 -12311.787} C_VEL
LIN {X 0,Y 376.186,Z 498.045,A -85,B 0,C 180,E1 -12314.004,E2 -12314.004} C_VEL
LIN {X 0,Y 375.465,Z 506.248,A -85,B 0,C 180,E1 -12316.22,E2 -12316.22} C_VEL
LIN {X 0,Y 374.985,Z 512.13,A -85,B 0,C 180,E1 -12318.102,E2 -12318.102} C_VEL
LIN {X 0,Y 374.69,Z 517.69,A -85,B 0,C 180,E1 -12320.281,E2 -12320.281} C_VEL
LIN {X 0,Y 374.707,Z 522.116,A -85,B 0,C 180,E1 -12322.455,E2 -12322.455} C_VEL
LIN {X 0,Y 374.8,Z 524,A -85,B 0,C 180,E1 -12323.625,E2 -12323.625} C_VEL
LIN {X 0,Y 374.678,Z 526.469,A -85,B 0,C 180,E1 -12325.696,E2 -12325.696} C_VEL
LIN {X 0,Y 374.828,Z 528.055,A -85,B 0,C 180,E1 -12327.85,E2 -12327.85} C_VEL
LIN {X 0,Y 374.86,Z 528.425,A -85,B 0,C 180,E1 -12329.999,E2 -12329.999} C_VEL
LIN {X 0,Y 374.844,Z 527.747,A -85,B 0,C 180,E1 -12332.148,E2 -12332.148} C_VEL
LIN {X 0,Y 374.846,Z 526.982,A -85,B 0,C 180,E1 -12333.224,E2 -12333.224} C_VEL
LIN {X 0,Y 374.778,Z 524.535,A -85,B 0,C 180,E1 -12335.379,E2 -12335.379} C_VEL
LIN {X 0,Y 374.77,Z 520.986,A -85,B 0,C 180,E1 -12337.542,E2 -12337.542} C_VEL
LIN {X 0,Y 374.754,Z 516.148,A -85,B 0,C 180,E1 -12339.716,E2 -12339.716} C_VEL
LIN {X 0,Y 375.017,Z 510.009,A -85,B 0,C 180,E1 -12341.896,E2 -12341.896} C_VEL
LIN {X 0,Y 375.491,Z 502.47,A -85,B 0,C 180,E1 -12344.082,E2 -12344.082} C_VEL
LIN {X 0,Y 376.239,Z 493.338,A -85,B 0,C 180,E1 -12346.271,E2 -12346.271} C_VEL
LIN {X 0,Y 377.063,Z 484.316,A -85,B 0,C 180,E1 -12348.089,E2 -12348.089} C_VEL
LIN {X 0,Y 378.299,Z 472.6,A -85,B 0,C 180,E1 -12350.101,E2 -12350.101} C_VEL
LIN {X 0,Y 379.772,Z 460.067,A -85,B 0,C 180,E1 -12351.916,E2 -12351.916} C_VEL
LIN {X 0,Y 381.38,Z 446.073,A -85,B 0,C 180,E1 -12353.628,E2 -12353.628} C_VEL
LIN {X 0,Y 383.061,Z 431.667,A -85,B 0,C 180,E1 -12355.104,E2 -12355.104} C_VEL
LIN {X 0,Y 384.666,Z 416.979,A -85,B 0,C 180,E1 -12356.365,E2 -12356.365} C_VEL
LIN {X 0,Y 386.364,Z 400.996,A -85,B 0,C 180,E1 -12357.488,E2 -12357.488} C_VEL
LIN {X 0,Y 387.843,Z 384.661,A -85,B 0,C 180,E1 -12358.402,E2 -12358.402} C_VEL
LIN {X 0,Y 389.098,Z 368.118,A -85,B 0,C 180,E1 -12359.113,E2 -12359.113} C_VEL
LIN {X 0,Y 390.137,Z 351.739,A -85,B 0,C 180,E1 -12359.62,E2 -12359.62} C_VEL
LIN {X 0,Y 396.608,Z 191.302,A -85,B 0,C 180,E1 -12363.396,E2 -12363.396} C_VEL
LIN {X 0,Y 392.088,Z 156.367,A -85,B 0,C 180,E1 -12364.686,E2 -12364.686} C_VEL
LIN {X 0,Y 388.148,Z 147.427,A -85,B 0,C 180,E1 -12365.266,E2 -12365.266} C_VEL
LIN {X 0,Y 383.085,Z 131.713,A -85,B 0,C 180,E1 -12367.615,E2 -12367.615} C_VEL
LIN {X 0,Y 376.838,Z 112.697,A -85,B 0,C 180,E1 -12370.613,E2 -12370.613} C_VEL
LIN {X 0,Y 375.996,Z 109.963,A -85,B 0,C 180,E1 -12371.08,E2 -12371.08} C_VEL
LIN {X 0,Y 375.974,Z 109.967,A -85,B 0,C 180,E1 -12374.739,E2 -12374.739} C_VEL
LIN {X 0,Y 375.93,Z 109.973,A -85,B 0,C 180,E1 -12378.399,E2 -12378.399} C_VEL
LIN {X 0,Y 375.971,Z 109.962,A -85,B 0,C 180,E1 -12381.729,E2 -12381.729} C_VEL
LIN {X 0,Y 375.975,Z 109.961,A -85,B 0,C 180,E1 -12385.332,E2 -12385.332} C_VEL
LIN {X 0,Y 375.971,Z 109.965,A -85,B 0,C 180,E1 -12388.44,E2 -12388.44} C_VEL
LIN {X 0,Y 375.998,Z 109.964,A -85,B 0,C 180,E1 -12392.142,E2 -12392.142} C_VEL
LIN {X 0,Y 376.001,Z 109.959,A -85,B 0,C 180,E1 -12394.539,E2 -12394.539} C_VEL
LIN {X 0,Y 375.958,Z 109.969,A -85,B 0,C 180,E1 -12398.046,E2 -12398.046} C_VEL
LIN {X 0,Y 376.019,Z 109.957,A -85,B 0,C 180,E1 -12401.474,E2 -12401.474} C_VEL
LIN {X 0,Y 376.058,Z 109.95,A -85,B 0,C 180,E1 -12404.833,E2 -12404.833} C_VEL
LIN {X 0,Y 376.054,Z 109.954,A -85,B 0,C 180,E1 -12408.137,E2 -12408.137} C_VEL
LIN {X 0,Y 376.253,Z 109.932,A -85,B 0,C 180,E1 -12411.877,E2 -12411.877} C_VEL
LIN {X 0,Y 376.167,Z 109.937,A -85,B 0,C 180,E1 -12414.64,E2 -12414.64} C_VEL
LIN {X 0,Y 376.349,Z 109.919,A -85,B 0,C 180,E1 -12417.86,E2 -12417.86} C_VEL
LIN {X 0,Y 376.484,Z 109.9,A -85,B 0,C 180,E1 -12420,E2 -12420} C_VEL
LIN {X 0,Y 376.185,Z 109.937,A -85,B 0,C 180,E1 -12423.213,E2 -12423.213} C_VEL
LIN {X 0,Y 376.23,Z 109.929,A -85,B 0,C 180,E1 -12426.628,E2 -12426.628} C_VEL
LIN {X 0,Y 376.201,Z 109.933,A -85,B 0,C 180,E1 -12428.595,E2 -12428.595} C_VEL
LIN {X 0,Y 376.046,Z 109.954,A -85,B 0,C 180,E1 -12431.864,E2 -12431.864} C_VEL
LIN {X 0,Y 376.054,Z 109.955,A -85,B 0,C 180,E1 -12435.168,E2 -12435.168} C_VEL
LIN {X 0,Y 376.004,Z 109.957,A -85,B 0,C 180,E1 -12438.527,E2 -12438.527} C_VEL
LIN {X 0,Y 375.959,Z 109.963,A -85,B 0,C 180,E1 -12441.955,E2 -12441.955} C_VEL
LIN {X 0,Y 376.002,Z 109.961,A -85,B 0,C 180,E1 -12445.461,E2 -12445.461} C_VEL
LIN {X 0,Y 375.957,Z 109.969,A -85,B 0,C 180,E1 -12449.08,E2 -12449.08} C_VEL
LIN {X 0,Y 375.945,Z 109.969,A -85,B 0,C 180,E1 -12452.829,E2 -12452.829} C_VEL
LIN {X 0,Y 375.954,Z 109.966,A -85,B 0,C 180,E1 -12455.416,E2 -12455.416} C_VEL
LIN {X 0,Y 375.972,Z 109.962,A -85,B 0,C 180,E1 -12458.271,E2 -12458.271} C_VEL
LIN {X 0,Y 375.931,Z 109.967,A -85,B 0,C 180,E1 -12461.601,E2 -12461.601} C_VEL
LIN {X 0,Y 375.952,Z 109.966,A -85,B 0,C 180,E1 -12465.265,E2 -12465.265} C_VEL
LIN {X 0,Y 375.978,Z 109.963,A -85,B 0,C 180,E1 -12469.139,E2 -12469.139} C_VEL
LIN {X 0,Y 375.962,Z 109.963,A -85,B 0,C 180,E1 -12471.912,E2 -12471.912} C_VEL
LIN {X 0,Y 375.977,Z 109.961,A -85,B 0,C 180,E1 -12475.333,E2 -12475.333} C_VEL
LIN {X 0,Y 375.955,Z 109.968,A -85,B 0,C 180,E1 -12478.439,E2 -12478.439} C_VEL
LIN {X 0,Y 375.981,Z 109.962,A -85,B 0,C 180,E1 -12482.141,E2 -12482.141} C_VEL
LIN {X 0,Y 376.005,Z 109.963,A -85,B 0,C 180,E1 -12484.54,E2 -12484.54} C_VEL
LIN {X 0,Y 375.97,Z 109.964,A -85,B 0,C 180,E1 -12488.047,E2 -12488.047} C_VEL
LIN {X 0,Y 376.029,Z 109.954,A -85,B 0,C 180,E1 -12491.475,E2 -12491.475} C_VEL
LIN {X 0,Y 376.058,Z 109.952,A -85,B 0,C 180,E1 -12494.833,E2 -12494.833} C_VEL
LIN {X 0,Y 376.05,Z 109.957,A -85,B 0,C 180,E1 -12498.137,E2 -12498.137} C_VEL
LIN {X 0,Y 376.258,Z 109.929,A -85,B 0,C 180,E1 -12501.878,E2 -12501.878} C_VEL
LIN {X 0,Y 376.171,Z 109.938,A -85,B 0,C 180,E1 -12504.641,E2 -12504.641} C_VEL
LIN {X 0,Y 376.352,Z 109.918,A -85,B 0,C 180,E1 -12507.86,E2 -12507.86} C_VEL
LIN {X 0,Y 376.488,Z 109.903,A -85,B 0,C 180,E1 -12510.001,E2 -12510.001} C_VEL
LIN {X 0,Y 376.186,Z 109.935,A -85,B 0,C 180,E1 -12513.214,E2 -12513.214} C_VEL
LIN {X 0,Y 376.248,Z 109.929,A -85,B 0,C 180,E1 -12516.436,E2 -12516.436} C_VEL
LIN {X 0,Y 376.207,Z 109.933,A -85,B 0,C 180,E1 -12518.596,E2 -12518.596} C_VEL
LIN {X 0,Y 376.052,Z 109.958,A -85,B 0,C 180,E1 -12521.864,E2 -12521.864} C_VEL
LIN {X 0,Y 376.06,Z 109.951,A -85,B 0,C 180,E1 -12525.168,E2 -12525.168} C_VEL
LIN {X 0,Y 376.011,Z 109.957,A -85,B 0,C 180,E1 -12528.527,E2 -12528.527} C_VEL
LIN {X 0,Y 375.965,Z 109.966,A -85,B 0,C 180,E1 -12531.955,E2 -12531.955} C_VEL
LIN {X 0,Y 376.009,Z 109.961,A -85,B 0,C 180,E1 -12535.462,E2 -12535.462} C_VEL
LIN {X 0,Y 375.963,Z 109.964,A -85,B 0,C 180,E1 -12539.08,E2 -12539.08} C_VEL
LIN {X 0,Y 375.952,Z 109.964,A -85,B 0,C 180,E1 -12542.829,E2 -12542.829} C_VEL
LIN {X 0,Y 375.96,Z 109.969,A -85,B 0,C 180,E1 -12545.416,E2 -12545.416} C_VEL
LIN {X 0,Y 375.977,Z 109.961,A -85,B 0,C 180,E1 -12548.271,E2 -12548.271} C_VEL
LIN {X 0,Y 375.985,Z 109.96,A -85,B 0,C 180,E1 -12550.032,E2 -12550.032} C_VEL
LIN {X 0,Y 375.253,Z 110.055,A -85,B 0,C 180,E1 -12550.925,E2 -12550.925} C_VEL
LIN {X 0,Y 372.346,Z 110.413,A -85,B 0,C 180,E1 -12552.377,E2 -12552.377} C_VEL
LIN {X 0,Y 369.943,Z 110.716,A -85,B 0,C 180,E1 -12553.552,E2 -12553.552} C_VEL
LIN {X 0,Y 368.948,Z 110.837,A -85,B 0,C 180,E1 -12554.46,E2 -12554.46} C_VEL
LIN {X 0,Y 368.885,Z 110.846,A -85,B 0,C 180,E1 -12554.768,E2 -12554.768} C_VEL
LIN {X 0,Y 368.885,Z 110.844,A -85,B 0,C 180,E1 -12558.178,E2 -12558.178} C_VEL
LIN {X 0,Y 368.911,Z 110.845,A -85,B 0,C 180,E1 -12561.36,E2 -12561.36} C_VEL
LIN {X 0,Y 368.959,Z 110.84,A -85,B 0,C 180,E1 -12563.887,E2 -12563.887} C_VEL
LIN {X 0,Y 370.104,Z 113.914,A -85,B 0,C 180,E1 -12564.099,E2 -12564.099} C_VEL
LIN {X 0,Y 386.532,Z 146.413,A -85,B 0,C 180,E1 -12566.388,E2 -12566.388} C_VEL
LIN {X 0,Y 389.785,Z 152.919,A -85,B 0,C 180,E1 -12566.816,E2 -12566.816} C_VEL
LIN {X 0,Y 383.64,Z 299.933,A -85,B 0,C 180,E1 -12570.355,E2 -12570.355} C_VEL
LIN {X 0,Y 382.762,Z 317.45,A -85,B 0,C 180,E1 -12570.997,E2 -12570.997} C_VEL
LIN {X 0,Y 381.524,Z 335.163,A -85,B 0,C 180,E1 -12571.877,E2 -12571.877} C_VEL
LIN {X 0,Y 380.199,Z 351.484,A -85,B 0,C 180,E1 -12572.922,E2 -12572.922} C_VEL
LIN {X 0,Y 378.674,Z 367.004,A -85,B 0,C 180,E1 -12574.142,E2 -12574.142} C_VEL
LIN {X 0,Y 377.065,Z 381.396,A -85,B 0,C 180,E1 -12575.499,E2 -12575.499} C_VEL
LIN {X 0,Y 375.431,Z 395.953,A -85,B 0,C 180,E1 -12577.143,E2 -12577.143} C_VEL
LIN {X 0,Y 373.958,Z 408.316,A -85,B 0,C 180,E1 -12578.791,E2 -12578.791} C_VEL
LIN {X 0,Y 372.645,Z 419.689,A -85,B 0,C 180,E1 -12580.561,E2 -12580.561} C_VEL
LIN {X 0,Y 371.277,Z 431.048,A -85,B 0,C 180,E1 -12582.654,E2 -12582.654} C_VEL
LIN {X 0,Y 370.169,Z 441.075,A -85,B 0,C 180,E1 -12584.867,E2 -12584.867} C_VEL
LIN {X 0,Y 369.411,Z 448.439,A -85,B 0,C 180,E1 -12586.803,E2 -12586.803} C_VEL
LIN {X 0,Y 368.725,Z 455.524,A -85,B 0,C 180,E1 -12589.012,E2 -12589.012} C_VEL
LIN {X 0,Y 368.345,Z 461.262,A -85,B 0,C 180,E1 -12591.22,E2 -12591.22} C_VEL
LIN {X 0,Y 368.061,Z 465.737,A -85,B 0,C 180,E1 -12593.421,E2 -12593.421} C_VEL
LIN {X 0,Y 367.873,Z 469.137,A -85,B 0,C 180,E1 -12595.617,E2 -12595.617} C_VEL
LIN {X 0,Y 367.924,Z 470.423,A -85,B 0,C 180,E1 -12596.715,E2 -12596.715} C_VEL
